// TIA Portal project "Mixing Fluid Projects" (V14)
// Project Files to accomodate the PLC Programming for Mixing Fluid Projects. 
// 
// PLEASE USE THE PROGRAM WISELY

(* hardware
DEVICE "S71500/ET200MP station_1"  S7-1500 station
   slot 0: "Rail_0"  Rack  6ES7 590-1***0-0AA0
   slot 0: "PS 60W 24/48/60VDC_1"  PS 60W 24/48/60VDC  6ES7 505-0RA00-0AB0  V1.0
   slot 1: "PLC_1"  CPU 1513-1 PN  6ES7 513-1AL01-0AB0  V2.1
      slot 3: "CPU display_1"  6ES7591-1AA00-0AA0
   slot 2: "DI 16x24VDC BA_1"  DI 16x24VDC BA  6ES7 521-1BH10-0AA0  V1.0
   slot 3: "DQ 16x24VDC/0.5A BA_1"  DQ 16x24VDC/0.5A BA  6ES7 522-1BH10-0AA0  V1.0
   slot 4: "AI 8xU/I/RTD/TC ST_1"  AI 8xU/I/RTD/TC ST  6ES7 531-7KF00-0AB0  V2.1
   slot 5: "AQ 8xU/I HS_1"  AQ 8xU/I HS  6ES7 532-5HF00-0AB0  V2.1
*)

// ===== PLC "PLC_1"  CPU 1513-1 PN =====

DATA_BLOCK "General_Tank Level_DB"   // DB4
{ S7_Optimized_Access := 'FALSE' }
VERSION : 0.1
   VAR
      "User Setpoint" : Int := 30;   // Setpoint Input from User
      PID_Level_Setpoint : Real;   // Setpoint into PID Level
      PID_Level_MV : Real;   // Output of PID Level (Manipulating Variable) on %
      PID_Level_MVNorm : Real;   // Output of PID Level (Manipulating Variable) on % Normalize
      PID_Level_MVInt : Int;   // Output of PID Level (Manipulating Variable) on % Integer
      PID_Level_ManualSlct : Bool;   // Switch for Activate Manual Mode
      PID_Level_InputMnlValue : Real;   // User Input Value for Manual MV
      PID_Level_ErrorAck : Bool;   // Acknowledged Button for Operator
      PID_Level_PIDReset : Bool;   // Reset Button for PID Compact
      PID_Level_ModeslctButton : Bool := true;   // Activate Mode Selection for PID Operation
      PID_Level_ModeValue : Int := 3;   // Select Mode for PID Operation from 1-4
      PID_Level_Alarm_SVHigh : Bool;   // Alarm from PID Level if Setpoint is Maximum
      PID_Level_Alarm_SVLow : Bool;   // Alarm from PID Level if Setpoint is Minimum
      PID_Level_Alarm_PVhigh : Bool;   // Alarm from PID Level if Process Value is Maximum
      PID_Level_Alarm_PVLow : Bool;   // Alarm from PID Level if Process Value is Minimum
      PID_Level_ModeStatus : Int;   // Status Mode for PID Operation
      PID_Level_ErrorStatus : Bool;   // Error Flag if PID Block is Occured
      PID_Level_ErrorBit : Real;   // Error Code if PID Block is Occured
      ControlValve_Level_Output : Real;   // Output of Level Control Valve
      ControlValve_Level_TravelMax : Bool;   // Level Control Valve Travel Max
      ControlValve_Level_TravelMin : Bool;   // Level Control Valve Travel Min
      "Level_Process Value" : Real := 50.0;   // Output from Level Process
      "Level_Process Reset" : Bool;   // Reset The Level Process
      Level_FlowarateAddRslt : Real;   // Additional PV from Hot + Cold Fluid Flowrate
      "Level_Flowrate Input" : Real;   // Total net flowrate going in/out from tank
      CascadeCommand : Bool;   // Command to activate Cascade PID Level Loop
      FeedforwardCmd : Bool;   // Command to activate Feedforward PID Level Loop
      LSH_Active : Bool;   // Alarm : Level Switch High Activate
      LSH_Warn : Bool;   // Alarm : Warning before LSH Active
      LSL_Active : Bool;   // Alarm : Level Switch Low Activate
      LSL_Warn : Bool;   // Alarm : Warning before LSL Active
      Trip_Reset : Bool := false;   // Alarm : Trip Command Reset
      PB_User : Real := 100.0;   // User Input for Proportional Band
      PB_UserDiv : Real := 0.0;   // User Input for Kp (Gain)
      Ti_User : Real := 104.7556;   // User Input for Integral Time
      Td_User : Real;   // User Input for Derivative Time
      SimpleFeedback_Status : Bool;   // Simple Feedback Loop Status Activate
   END_VAR
BEGIN
END_DATA_BLOCK

DATA_BLOCK "General_Flow Product 13_DB"   // DB5
{ S7_Optimized_Access := 'FALSE' }
VERSION : 0.1
   VAR
      User_Setpoint : Real := 2.0;   // Setpoint Input from User
      User_Setpoint_Norm : Real;   // Setpoint Input from User Normalized
      PID_Flow13_Setpoint : Real;   // Setpoint into PID Product Flowrate 13
      PID_Flow13_MV : Real;   // Output of PID Product Flowrate 13(Manipulating Variable) on %
      PID_Flow13_MVNorm : Real;   // Output of PID Product Flowrate 13(Manipulating Variable) on % Normalize
      PID_Flow13_MVInt : Int;   // Output of PID Product Flowrate 13 (Manipulating Variable) on % Integer
      PID_Flow13_ManualSlct : Bool;   // Switch for Activate Manual Mode
      PID_Flow13_InputMnlValue : Real;   // User Input Value for Manual MV
      PID_Flow13_ErrorAck : Bool;   // Acknowledged Button for Operator
      PID_Flow13_PIDReset : Bool;   // Reset Button for PID Compact
      PID_Flow13_ModeslctButton : Bool := true;   // Activate Mode Selection for PID Operation
      PID_Flow13_ModeValue : Int := 3;   // Select Mode for PID Operation from 1-4
      PID_Flow13_Alarm_SVHigh : Bool;   // Alarm from PID Product Flowrate 13 if Setpoint is Maximum
      PID_Flow13_Alarm_SVLow : Bool;   // Alarm from PID Product Flowrate 13 if Setpoint is Minimum
      PID_Flow13_Alarm_PVhigh : Bool;   // Alarm from PID Product Flowrate 13 if Process Value is Maximum
      PID_Flow13_Alarm_PVLow : Bool;   // Alarm from PID Product Flowrate 13 if Process Value is Minimum
      PID_Flow13_ModeStatus : Int;   // Status Mode for PID Operation
      PID_Flow13_ErrorStatus : Bool;   // Error Flag if PID Block is Occured
      PID_Flow13_ErrorBit : Real;   // Error Code if PID Block is Occured
      ControlValve_Flow13_Output : Real;   // Output of Product Flowrate 13 Control Valve
      ControlValve_Flow13_TravelMax : Bool;   // Product Flowrate 13 Control Valve Travel Max
      ControlValve_Flow13_TravelMin : Bool;   // Product Flowrate 13 Control Valve Travel Min
      "Flow13_Process Value" : Real;   // Output from Product Flowrate 13 Process
      "Flow13_Process ValueNorm" : Real;   // Output fromProduct Flowrate 13 Process Normalize
      "Flow13_Process Value_Status" : Real;   // Output Status from Product Flowrate
      "Flow13_Process Reset" : Bool;   // Reset The Product Flowrate 13Process
      SDV13_Active : Bool;   // Alarm : SDV13 Activate
      Pump13_CmdOffTrip : Bool;   // Turn off the Pump1-3 as Alarm Occured
      Pump13_CmdOff : Bool;   // Turn off the Pump1-3
      Pump13_CmdOn : Bool := false;   // Turn On the Pump1-3
      Pump13_Running : Bool := true;   // Pump1-3 Running Status
      Pump13_TripStatus : Bool;   // Pump1-3 Trip Status
      Pump13_TripReset : Bool := false;   // Pump1-3 Trip Reset Command
      PSL13_Active : Bool;   // Alarm : PSL Activate
      PSH13_Active : Bool;   // Alarm : PSH Activate
      PSH13_Reset : Bool;   // Reset Command of PSH13
      PB_User : Real := 21.71176;   // User Input for Proportional Band
      PB_UserDiv : Real;   // User Input for Kp (Gain)
      Ti_User : Real := 4.404553;   // User Input for Integral Time
      Td_User : Real := 0.0;   // User Input for Derivative Time
   END_VAR
BEGIN
END_DATA_BLOCK

DATA_BLOCK "General_Product Temperature_DB"   // DB9
{ S7_Optimized_Access := 'FALSE' }
VERSION : 0.1
   VAR
      User_Setpoint : Int := 40;   // Setpoint Input from User
      User_Setpoint_Norm : Real;   // Setpoint Input from User Normalized
      PID_Temp_Setpoint : Real;   // Setpoint into PID Product Temperature
      PID_Temp_MV : Real;   // Output of PID Product Temperature(Manipulating Variable) on %
      PID_Temp_MVNorm : Real;   // Output of PID Product Temperature(Manipulating Variable) on % Normalize
      PID_Temp_MVInt : Int;   // Output of PID Product Temperature (Manipulating Variable) on % Integer
      PID_Temp_ManualSlct : Bool;   // Switch for Activate Manual Mode
      PID_Temp_InputMnlValue : Real;   // User Input Value for Manual MV
      PID_Temp_ErrorAck : Bool;   // Acknowledged Button for Operator
      PID_Temp_PIDReset : Bool;   // Reset Button for PID Compact
      PID_Temp_ModeslctButton : Bool := true;   // Activate Mode Selection for PID Operation
      PID_Temp_ModeValue : Int := 3;   // Select Mode for PID Operation from 1-4
      PID_Temp_Alarm_SVHigh : Bool;   // Alarm from PID Product Temperature if Setpoint is Maximum
      PID_Temp_Alarm_SVLow : Bool;   // Alarm from PID Product Temperature if Setpoint is Minimum
      PID_Temp_Alarm_PVhigh : Bool;   // Alarm from PID Product Temperature if Process Value is Maximum
      PID_Temp_Alarm_PVLow : Bool;   // Alarm from PID Product Temperature if Process Value is Minimum
      PID_Temp_ModeStatus : Int;   // Status Mode for PID Operation
      PID_Temp_ErrorStatus : Bool;   // Error Flag if PID Block is Occured
      PID_Temp_ErrorBit : Real;   // Error Code if PID Block is Occured
      ControlValve_Temp_Output : Real;   // Output of Product Temperature Control Valve
      ControlValve_Temp_TravelMax : Bool;   // Product Temperature Control Valve Travel Max
      ControlValve_Temp_TravelMin : Bool;   // Product Temperature Control Valve Travel Min
      "Temp_Process Value" : Real;   // Output from Product Temperature Process
      "Temp_Process ValueRaw" : Real := 50.0;   // Output from Product Temperature Process raw
      "Temp_Process ValueNorm" : Real;   // Output fromProduct Temperature Process Normalize
      "Temp_Process Value_Status" : Real;   // Output Status from Product Temperature
      "Temp_Process Reset" : Bool;   // Reset The Product TemperatureProcess
      BlackCalc_HotFluid1Calc : Real;   // Hot Fluid Aspect Flowarate Heat released
      BlackCalc_ColdFluid1Calc_1 : Real;   // Hot Fluid Aspect Flowarate Heat received
      BlackCalc_Nominator : Real;   // Total additional of Black Calculation in Nominator
      BlackCalc_HotFluidFlowrate : Real;   // Flowrate of Hot Fluid in System
      BlackCalc_denominator : Real;   // Total additional of Black Calculation in denominator
      CascadeCmd : Bool;   // Cascade Command between Temp Product - Cold Fluid Flowrate
      FeedforwardCmd : Bool;   // Feedforward Command for Product Temp Control
      TSH_active : Bool;   // Alarm : Temp Switch High Activate
      TSH_Warn : Bool;   // Alarm : Warning before TSH Active
      TSL_active : Bool;   // Alarm : Temp Switch Low Activate
      TSL_Warn : Bool;   // Alarm : Warning before LSL Active
      Trip_Reset : Bool := false;   // Alarm : Trip Command Reset
      PB_User : Real := 50.0;   // User Input for Proportional Band
      PB_UserDiv : Real;   // User Input for Kp (Gain)
      Ti_User : Real := 4.404553;   // User Input for Integral Time
      Td_User : Real := 0.0;   // User Input for Derivative Time
      SimpleFeedback_Status : Bool;   // Simple Feedback Loop Status Activate
   END_VAR
BEGIN
END_DATA_BLOCK

DATA_BLOCK "General_Hot Fluid Flow_DB"   // DB12
{ S7_Optimized_Access := 'FALSE' }
VERSION : 0.1
   VAR
      User_Setpoint : Real := 2.5;   // Setpoint Input from User
      User_Setpoint_Norm : Real;   // Setpoint Input from User Normalized
      PID_Flow11_Setpoint : Real;   // Setpoint into PID Hot Fluid Flowrate
      PID_Flow11_MV : Real;   // Output of PIDHot Fluid Flowrate(Manipulating Variable) on %
      PID_Flow11_MVNorm : Real;   // Output of PID Hot Fluid Flowrate(Manipulating Variable) on % Normalize
      PID_Flow11_MVInt : Int;   // Output of PID Hot Fluid Flowrate (Manipulating Variable) on % Integer
      PID_Flow11_ManualSlct : Bool;   // Switch for Activate Manual Mode
      PID_Flow11_InputMnlValue : Real;   // User Input Value for Manual MV
      PID_Flow11_ErrorAck : Bool;   // Acknowledged Button for Operator
      PID_Flow11_PIDReset : Bool;   // Reset Button for PID Compact
      PID_Flow11_ModeslctButton : Bool := true;   // Activate Mode Selection for PID Operation
      PID_Flow11_ModeValue : Int := 3;   // Select Mode for PID Operation from 1-4
      PID_Flow11_Alarm_SVHigh : Bool;   // Alarm from PID Hot Fluid Flowrate if Setpoint is Maximum
      PID_Flow11_Alarm_SVLow : Bool;   // Alarm from PID Hot Fluid Flowrate if Setpoint is Minimum
      PID_Flow11_Alarm_PVhigh : Bool;   // Alarm from PID Hot Fluid Flowrate if Process Value is Maximum
      PID_Flow11_Alarm_PVLow : Bool;   // Alarm from PID Hot Fluid Flowrate if Process Value is Minimum
      PID_Flow11_ModeStatus : Int;   // Status Mode for PID Operation
      PID_Flow11_ErrorStatus : Bool;   // Error Flag if PID Block is Occured
      PID_Flow11_ErrorBit : Real;   // Error Code if PID Block is Occured
      ControlValve_Flow11_Output : Real;   // Output of Hot Fluid Flowrate Control Valve
      ControlValve_Flow11_TravelMax : Bool;   // Product Hot Fluid Flowrate Control Valve Travel Max
      ControlValve_Flow11_TravelMin : Bool;   // Product Hot Fluid Flowrate Control Valve Travel Min
      "Flow11_Process Value" : Real;   // Output from Hot Fluid Flowrate Process
      "Flow11_Process ValueNorm" : Real;   // Output fromHot Fluid Flowrate Process Normalize
      "Flow11_Process Value_Status" : Real;   // Output Status from Hot Fluid Flowrate
      "Flow11_Process Reset" : Bool;   // Reset The Hot Fluid Flowrate Process
      Flow11_LoopActv : Bool := true;   // Command to activate Hot Fluid Control Loop Only
      SDV11_Active : Bool;   // Alarm : SDV11_Activate
      Pump11_CmdOffTrip : Bool;   // Turn Off the Pump1-1 as Alarm Activate
      Pump11_CmdOff : Bool;   // Turn off the Pump1-1
      Pump11_CmdOn : Bool := false;   // Turn On the Pump1-1
      Pump11_Running : Bool := true;   // Pump1-1 Running Status
      Pump11_TripStatus : Bool;   // Pump1-1 Trip Status
      Pump11_TripReset : Bool := false;   // Pump1-1 Trip Reset Command
      PSL11_Active : Bool;   // Alarm : PSL Activate
      PSH11_Active : Bool;   // Alarm : PSH Activate
      PSH11_Reset : Bool := false;   // Reset Command of PSH11
      PB_User : Real := 100.0;   // User Input for Proportional Band
      PB_UserDiv : Real;   // User Input for Kp (Gain)
      Ti_User : Real := 20.0;   // User Input for Integral Time
      Td_User : Real;   // User Input for Derivative Time
   END_VAR
BEGIN
END_DATA_BLOCK

DATA_BLOCK "General_Cold Fluid Flow_DB"   // DB15
{ S7_Optimized_Access := 'FALSE' }
VERSION : 0.1
   VAR
      User_Setpoint : Real := 1.7;   // Setpoint Input from User
      User_Setpoint_Norm : Real;   // Setpoint Input from User Normalized
      PID_Flow12_Setpoint : Real;   // Setpoint into PID Cold Fluid Flowrate
      PID_Flow12_MV : Real;   // Output of PID Cold Fluid Flowrate(Manipulating Variable) on %
      PID_Flow12_MVNorm : Real;   // Output of PID Cold Fluid Flowrate(Manipulating Variable) on % Normalize
      PID_Flow12_MVInt : Int;   // Output of PID Cold Fluid Flowrate (Manipulating Variable) on % Integer
      PID_Flow12_ManualSlct : Bool;   // Switch for Activate Manual Mode
      PID_Flow12_InputMnlValue : Real;   // User Input Value for Manual MV
      PID_Flow12_ErrorAck : Bool;   // Acknowledged Button for Operator
      PID_Flow12_PIDReset : Bool;   // Reset Button for PID Compact
      PID_Flow12_ModeslctButton : Bool := true;   // Activate Mode Selection for PID Operation
      PID_Flow12_ModeValue : Int := 3;   // Select Mode for PID Operation from 1-4
      PID_Flow12_Alarm_SVHigh : Bool;   // Alarm from PID Cold Fluid Flowrate if Setpoint is Maximum
      PID_Flow12_Alarm_SVLow : Bool;   // Alarm from PID Cold Fluid Flowrate if Setpoint is Minimum
      PID_Flow12_Alarm_PVhigh : Bool;   // Alarm from PID ColdFluid Flowrate if Process Value is Maximum
      PID_Flow12_Alarm_PVLow : Bool;   // Alarm from PID Cold Fluid Flowrate if Process Value is Minimum
      PID_Flow12_ModeStatus : Int;   // Status Mode for PID Operation
      PID_Flow12_ErrorStatus : Bool;   // Error Flag if PID Block is Occured
      PID_Flow12_ErrorBit : Real;   // Error Code if PID Block is Occured
      ControlValve_Flow12_Output : Real;   // Output of Cold Fluid Flowrate Control Valve
      ControlValve_Flow12_TravelMax : Bool;   // Product Cold Fluid Flowrate Control Valve Travel Max
      ControlValve_Flow12_TravelMin : Bool;   // Product Cold Fluid Flowrate Control Valve Travel Min
      "Flow12_Process Value" : Real;   // Output from Cold Fluid Flowrate Process
      "Flow12_Process ValueNorm" : Real;   // Output from Cold Fluid Flowrate Process Normalize
      "Flow12_Process Value_Status" : Real;   // Output Status from Cold Fluid Flowrate
      "Flow12_Process Reset" : Bool;   // Reset The Cold Fluid Flowrate Process
      Flow12_LoopActv : Bool := true;   // Activate the Cold Fluid Control Loop Only
      SDV12_Active : Bool;   // Alarm : SDV12 activate
      Pump12_CmdOffTrip : Bool;   // Turn Off the Pump1-2 as Alarm Occured
      Pump12_CmdOff : Bool;   // Turn off the Pump1-2
      Pump12_CmdOn : Bool := false;   // Turn On the Pump1-2
      Pump12_Running : Bool := true;   // Pump1-2 Running Status
      Pump12_TripStatus : Bool;   // Pump1-2 Trip Status
      Pump12_TripReset : Bool := false;   // Pump1-2 Trip Reset Command
      PSL12_Active : Bool;   // Alarm : PSL Activate
      PSH12_Active : Bool;   // Alarm : PSH Activate
      PSH12_Reset : Bool;   // Reset Command of PSH12
      PB_User : Real := 21.56999;   // User Input for Proportional Band
      PB_UserDiv : Real;   // User Input for Kp (Gain)
      Ti_User : Real := 4.443021;   // User Input for Integral Time
      Td_User : Real := 0.0;   // User Input for Derivative Time
   END_VAR
BEGIN
END_DATA_BLOCK

// folder: Alarm Group DB

DATA_BLOCK "Program Alarm_DB_LSH"   // DB22
{ S7_Optimized_Access := 'TRUE' }
VERSION : 0.1
// stored: InstanceOfName Program Alarm
"Program Alarm"
BEGIN
END_DATA_BLOCK

DATA_BLOCK "Program Alarm_DB_LSL"   // DB23
{ S7_Optimized_Access := 'TRUE' }
VERSION : 0.1
// stored: InstanceOfName Program Alarm
"Program Alarm"
BEGIN
END_DATA_BLOCK

DATA_BLOCK "Program Alarm Unack_DB_LSHWarn"   // DB24
{ S7_Optimized_Access := 'TRUE' }
VERSION : 0.1
// stored: InstanceOfName Program Alarm Unack
"Program Alarm Unack"
BEGIN
END_DATA_BLOCK

DATA_BLOCK "Program Alarm Unack_DB_LSLWarn"   // DB25
{ S7_Optimized_Access := 'TRUE' }
VERSION : 0.1
// stored: InstanceOfName Program Alarm Unack
"Program Alarm Unack"
BEGIN
END_DATA_BLOCK

DATA_BLOCK "Program Alarm_DB_TSH"   // DB26
{ S7_Optimized_Access := 'TRUE' }
VERSION : 0.1
// stored: InstanceOfName Program Alarm
"Program Alarm"
BEGIN
END_DATA_BLOCK

DATA_BLOCK "Program Alarm Unack_DB_TSHWarn"   // DB27
{ S7_Optimized_Access := 'TRUE' }
VERSION : 0.1
// stored: InstanceOfName Program Alarm Unack
"Program Alarm Unack"
BEGIN
END_DATA_BLOCK

DATA_BLOCK "Program Alarm_DB_TSL"   // DB28
{ S7_Optimized_Access := 'TRUE' }
VERSION : 0.1
// stored: InstanceOfName Program Alarm
"Program Alarm"
BEGIN
END_DATA_BLOCK

DATA_BLOCK "Program Alarm Unack_DB_TSLWarn"   // DB29
{ S7_Optimized_Access := 'TRUE' }
VERSION : 0.1
// stored: InstanceOfName Program Alarm Unack
"Program Alarm Unack"
BEGIN
END_DATA_BLOCK

DATA_BLOCK "Program Alarm_DB_PSH11"   // DB30
{ S7_Optimized_Access := 'TRUE' }
VERSION : 0.1
// stored: InstanceOfName Program Alarm
"Program Alarm"
BEGIN
END_DATA_BLOCK

DATA_BLOCK "Program Alarm_DB_SDV11"   // DB31
{ S7_Optimized_Access := 'TRUE' }
VERSION : 0.1
// stored: InstanceOfName Program Alarm
"Program Alarm"
BEGIN
END_DATA_BLOCK

DATA_BLOCK "Program Alarm_DB_Pump11TripStatus"   // DB32
{ S7_Optimized_Access := 'TRUE' }
VERSION : 0.1
// stored: InstanceOfName Program Alarm
"Program Alarm"
BEGIN
END_DATA_BLOCK

DATA_BLOCK "Program Alarm Unack_DB_Pump11Run"   // DB33
{ S7_Optimized_Access := 'TRUE' }
VERSION : 0.1
// stored: InstanceOfName Program Alarm Unack
"Program Alarm Unack"
BEGIN
END_DATA_BLOCK

DATA_BLOCK "Program Alarm Unack_DB_Pump11CmdOff"   // DB34
{ S7_Optimized_Access := 'TRUE' }
VERSION : 0.1
// stored: InstanceOfName Program Alarm Unack
"Program Alarm Unack"
BEGIN
END_DATA_BLOCK

DATA_BLOCK "Program Alarm Unack_DB_Pump11TripReset"   // DB35
{ S7_Optimized_Access := 'TRUE' }
VERSION : 0.1
// stored: InstanceOfName Program Alarm Unack
"Program Alarm Unack"
BEGIN
END_DATA_BLOCK

DATA_BLOCK "Program Alarm Unack_DB_PSL11"   // DB36
{ S7_Optimized_Access := 'TRUE' }
VERSION : 0.1
// stored: InstanceOfName Program Alarm Unack
"Program Alarm Unack"
BEGIN
END_DATA_BLOCK

DATA_BLOCK "Program Alarm Unack_DB_PSH11Reset"   // DB37
{ S7_Optimized_Access := 'TRUE' }
VERSION : 0.1
// stored: InstanceOfName Program Alarm Unack
"Program Alarm Unack"
BEGIN
END_DATA_BLOCK

DATA_BLOCK "Program Alarm_DB_PSH12"   // DB38
{ S7_Optimized_Access := 'TRUE' }
VERSION : 0.1
// stored: InstanceOfName Program Alarm
"Program Alarm"
BEGIN
END_DATA_BLOCK

DATA_BLOCK "Program Alarm_DB_SDV12"   // DB39
{ S7_Optimized_Access := 'TRUE' }
VERSION : 0.1
// stored: InstanceOfName Program Alarm
"Program Alarm"
BEGIN
END_DATA_BLOCK

DATA_BLOCK "Program Alarm_DB_Pump12TripStatus"   // DB40
{ S7_Optimized_Access := 'TRUE' }
VERSION : 0.1
// stored: InstanceOfName Program Alarm
"Program Alarm"
BEGIN
END_DATA_BLOCK

DATA_BLOCK "Program Alarm Unack_DB_Pump12Run"   // DB41
{ S7_Optimized_Access := 'TRUE' }
VERSION : 0.1
// stored: InstanceOfName Program Alarm Unack
"Program Alarm Unack"
BEGIN
END_DATA_BLOCK

DATA_BLOCK "Program Alarm Unack_DB_Pump12CmdOff"   // DB42
{ S7_Optimized_Access := 'TRUE' }
VERSION : 0.1
// stored: InstanceOfName Program Alarm Unack
"Program Alarm Unack"
BEGIN
END_DATA_BLOCK

DATA_BLOCK "Program Alarm Unack_DB_Pump12TripReset"   // DB43
{ S7_Optimized_Access := 'TRUE' }
VERSION : 0.1
// stored: InstanceOfName Program Alarm Unack
"Program Alarm Unack"
BEGIN
END_DATA_BLOCK

DATA_BLOCK "Program Alarm Unack_DB_PSL12"   // DB44
{ S7_Optimized_Access := 'TRUE' }
VERSION : 0.1
// stored: InstanceOfName Program Alarm Unack
"Program Alarm Unack"
BEGIN
END_DATA_BLOCK

DATA_BLOCK "Program Alarm Unack_DB_PSH12Reset"   // DB45
{ S7_Optimized_Access := 'TRUE' }
VERSION : 0.1
// stored: InstanceOfName Program Alarm Unack
"Program Alarm Unack"
BEGIN
END_DATA_BLOCK

DATA_BLOCK "Program Alarm_DB_PSH13"   // DB46
{ S7_Optimized_Access := 'TRUE' }
VERSION : 0.1
// stored: InstanceOfName Program Alarm
"Program Alarm"
BEGIN
END_DATA_BLOCK

DATA_BLOCK "Program Alarm_DB_SDV13"   // DB47
{ S7_Optimized_Access := 'TRUE' }
VERSION : 0.1
// stored: InstanceOfName Program Alarm
"Program Alarm"
BEGIN
END_DATA_BLOCK

DATA_BLOCK "Program Alarm_DB_Pump13TripStatus"   // DB48
{ S7_Optimized_Access := 'TRUE' }
VERSION : 0.1
// stored: InstanceOfName Program Alarm
"Program Alarm"
BEGIN
END_DATA_BLOCK

DATA_BLOCK "Program Alarm Unack_DB_Pump13Run"   // DB49
{ S7_Optimized_Access := 'TRUE' }
VERSION : 0.1
// stored: InstanceOfName Program Alarm Unack
"Program Alarm Unack"
BEGIN
END_DATA_BLOCK

DATA_BLOCK "Program Alarm Unack_DB_Pump13CmdOff"   // DB50
{ S7_Optimized_Access := 'TRUE' }
VERSION : 0.1
// stored: InstanceOfName Program Alarm Unack
"Program Alarm Unack"
BEGIN
END_DATA_BLOCK

DATA_BLOCK "Program Alarm Unack_DB_Pump13TripReset"   // DB51
{ S7_Optimized_Access := 'TRUE' }
VERSION : 0.1
// stored: InstanceOfName Program Alarm Unack
"Program Alarm Unack"
BEGIN
END_DATA_BLOCK

DATA_BLOCK "Program Alarm Unack_DB-PSL13"   // DB52
{ S7_Optimized_Access := 'TRUE' }
VERSION : 0.1
// stored: InstanceOfName Program Alarm Unack
"Program Alarm Unack"
BEGIN
END_DATA_BLOCK

DATA_BLOCK "Program Alarm Unack_DB_PSH13Reset"   // DB53
{ S7_Optimized_Access := 'TRUE' }
VERSION : 0.1
// stored: InstanceOfName Program Alarm Unack
"Program Alarm Unack"
BEGIN
END_DATA_BLOCK

DATA_BLOCK "Program Alarm Unack_DB_Level_Alarm Reset"   // DB54
{ S7_Optimized_Access := 'TRUE' }
VERSION : 0.1
// stored: InstanceOfName Program Alarm Unack
"Program Alarm Unack"
BEGIN
END_DATA_BLOCK

DATA_BLOCK "Program Alarm Unack_DB_Temp_Trip Reset"   // DB55
{ S7_Optimized_Access := 'TRUE' }
VERSION : 0.1
// stored: InstanceOfName Program Alarm Unack
"Program Alarm Unack"
BEGIN
END_DATA_BLOCK

// folder: System blocks/Program resources

DATA_BLOCK "Time On Delay PSH11"   // DB18
{ S7_Optimized_Access := 'TRUE' }
AUTHOR : Simatic
FAMILY : IEC
NAME : IEC_TMR
VERSION : 1.0
// stored: InstanceOfName IEC_TIMER
"IEC_TIMER"
BEGIN
END_DATA_BLOCK

DATA_BLOCK "Time On Delay PSH12"   // DB19
{ S7_Optimized_Access := 'TRUE' }
AUTHOR : Simatic
FAMILY : IEC
NAME : IEC_TMR
VERSION : 1.0
// stored: InstanceOfName IEC_TIMER
"IEC_TIMER"
BEGIN
END_DATA_BLOCK

DATA_BLOCK "Time On Delay PSH13"   // DB20
{ S7_Optimized_Access := 'TRUE' }
AUTHOR : Simatic
FAMILY : IEC
NAME : IEC_TMR
VERSION : 1.0
// stored: InstanceOfName IEC_TIMER
"IEC_TIMER"
BEGIN
END_DATA_BLOCK

DATA_BLOCK "TON_LSH"   // DB21
{ S7_Optimized_Access := 'TRUE' }
AUTHOR : Simatic
FAMILY : IEC
NAME : IEC_LTMR
VERSION : 1.0
// stored: InstanceOfName IEC_LTIMER
"IEC_LTIMER"
BEGIN
END_DATA_BLOCK

DATA_BLOCK "TON_LSL"   // DB56
{ S7_Optimized_Access := 'TRUE' }
AUTHOR : Simatic
FAMILY : IEC
NAME : IEC_LTMR
VERSION : 1.0
// stored: InstanceOfName IEC_LTIMER
"IEC_LTIMER"
BEGIN
END_DATA_BLOCK

DATA_BLOCK "TON_TSH"   // DB57
{ S7_Optimized_Access := 'TRUE' }
AUTHOR : Simatic
FAMILY : IEC
NAME : IEC_LTMR
VERSION : 1.0
// stored: InstanceOfName IEC_LTIMER
"IEC_LTIMER"
BEGIN
END_DATA_BLOCK

DATA_BLOCK "TON_TSL"   // DB58
{ S7_Optimized_Access := 'TRUE' }
AUTHOR : Simatic
FAMILY : IEC
NAME : IEC_TMR
VERSION : 1.0
// stored: InstanceOfName IEC_TIMER
"IEC_TIMER"
BEGIN
END_DATA_BLOCK

// folder: Utilities Group DB

DATA_BLOCK "Level Control Valve_DB"   // DB2
{ S7_Optimized_Access := 'TRUE' }
VERSION : 2.01
// stored: InstanceOfName LSim_Level Control Valve
"LSim_Level Control Valve"
BEGIN
   perOn := true;
END_DATA_BLOCK

DATA_BLOCK "LSim_Tank Process_DB"   // DB3
{ S7_Optimized_Access := 'TRUE' }
VERSION : 2.01
// stored: InstanceOfName LSim_Level Process
"LSim_Level Process"
BEGIN
END_DATA_BLOCK

DATA_BLOCK "Flow Control Valve 13_DB"   // DB7
{ S7_Optimized_Access := 'TRUE' }
VERSION : 2.01
// stored: InstanceOfName LSim_Flow Control Valve 13
"LSim_Flow Control Valve 13"
BEGIN
   perOn := true;
END_DATA_BLOCK

DATA_BLOCK "LSim_Product Flow 13 Process_DB"   // DB8
{ S7_Optimized_Access := 'TRUE' }
VERSION : 2.01
// stored: InstanceOfName LSim_Product Flowrate 13
"LSim_Product Flowrate 13"
BEGIN
END_DATA_BLOCK

DATA_BLOCK "LSim_Product Temp_DB"   // DB11
{ S7_Optimized_Access := 'TRUE' }
VERSION : 2.01
// stored: InstanceOfName LSim_Product Temp
"LSim_Product Temp"
BEGIN
   perOn := true;
END_DATA_BLOCK

DATA_BLOCK "LSim_Hot Fluid Flow_DB"   // DB14
{ S7_Optimized_Access := 'TRUE' }
VERSION : 2.01
// stored: InstanceOfName LSim_Hot Fluid Flowrate
"LSim_Hot Fluid Flowrate"
BEGIN
END_DATA_BLOCK

DATA_BLOCK "LSim_Cold Fluid Flowrate"   // DB17
{ S7_Optimized_Access := 'TRUE' }
VERSION : 2.01
// stored: InstanceOfName LSim_Cold Fluid Flow
"LSim_Cold Fluid Flow"
BEGIN
END_DATA_BLOCK

// folder: (top level)

FUNCTION_BLOCK "LSim_Flow Control Valve 13"   // FB1, FBD
{ S7_Optimized_Access := 'TRUE' }
VERSION : 2.01
// //============================================================================
// //SIEMENS AG
// //(c)Copyright 2017 All Rights Reserved
// //-----------------------------------------------------------------------------
// //Library:       Library for Controlled System Simulation
// //Tested with:   S7-1500 FW V2.0 / S7-1200 FW V4.2
// //Engineering:   STEP 7 V14 Upd2 (TIA Portal)
// //Restrictions:  Cyclic interrupt
// //Requirements:  memory card needed for S7-1500
// //Functionality: Simulation of a valve with adjustable transition time
// //-----------------------------------------------------------------------------
// //Change log table:
// //Version    Date             Expert in charge                               Changes applied
// //02.00.00 03.02.2016 Siemens Industry Online Support Release (STEP 7 V13 SP1)
// //02.00.01 02.03.2017 Siemens Industry Online Support Release (STEP 7 V14)
// //============================================================================
   VAR_INPUT
      inputUp : Bool := false;   // control signal “Open valve”
      inputDn : Bool := false;   // control signal “Close valve”
      inputPer : Int;   // Analog manipulated variable
      perOn : Bool;   // selection switch, whether inputUp/inputDn or inputPer is used (inputPer is used for TRUE)
      perMax : Real := 27648.0;   // upper limit of the analog value of the valve position.
      perMin : Real;   // lower limit of the analog value of the valve position
      realMax : Real := 100.0;   // upper limit of the converted floating-point value for the valve position
      realMin : Real;   // lower limit of the converted floating-point value for the valve position
      transitTime : Real := 20.0;   // traversing time of the value between the end positions
      cycle : Real := 0.1;   // cyclic time [sec]
      reset : Bool := false;   // resets all relevant parameters to ‘0’ including the output
   END_VAR
   VAR_OUTPUT
      output : Real := 0.0;   // calculated valve position (within the “realMin” and “realMax” limits)
      outputPer : Int;   // calculated analog valve position (within the “perMin” and “perMax” limits)
      highLimit : Bool := false;   // simulated upper valve end position reached at highLimit = TRUE
      lowLimit : Bool := false;   // simulated lower valve end position reached at lowLimit = TRUE
   END_VAR
   VAR
      statInput : Real;
      statDelta : Real;
      statOut : Real;
      statHigh : Bool;
      statLow : Bool;
   END_VAR
   VAR_TEMP
      tempReal : Real;
      tempStepWidth : Real;
      tempStepWidthNeg : Real;
      tempBool : Bool;
      tempInputNorm : Real;
      tempUpFlag : Bool;
      tempDnFlag : Bool;
      tempInt : Int;
   END_VAR
   VAR_TEMP   // added for the SCL form of the ladder/FBD networks
      _w1 : Bool;
   END_VAR
BEGIN

REGION Network 1: reset
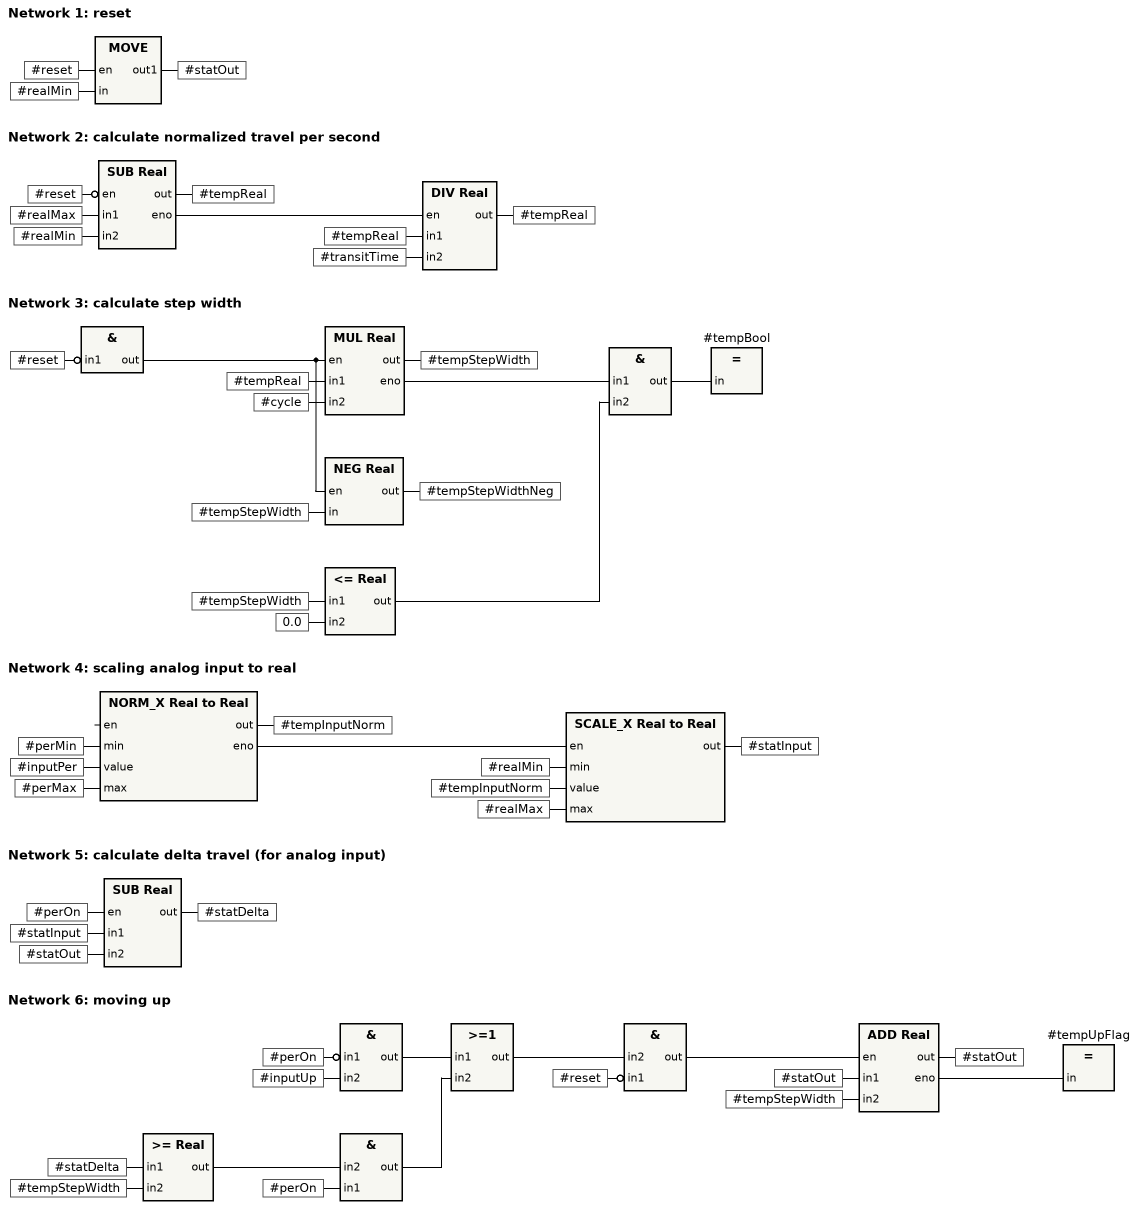
   IF #reset THEN #statOut := #realMin; END_IF;
END_REGION

REGION Network 2: calculate normalized travel per second
   // ENO of a box is taken as its EN; it also drops when the box reports an error
   IF NOT #reset THEN
       #tempReal := #realMax - #realMin;
       #tempReal := #tempReal / #transitTime;
   END_IF;
END_REGION

REGION Network 3: calculate step width
   // ENO of a box is taken as its EN; it also drops when the box reports an error
   IF NOT #reset THEN #tempStepWidth := #tempReal * #cycle; END_IF;
   #tempBool := NOT #reset AND (#tempStepWidth <= 0.0);
   IF NOT #reset THEN #tempStepWidthNeg := -#tempStepWidth; END_IF;
END_REGION

REGION Network 4: scaling analog input to real
   // ENO of a box is taken as its EN; it also drops when the box reports an error
   #tempInputNorm := NORM_X(MIN := #perMin, VALUE := #inputPer, MAX := #perMax);
   #statInput := SCALE_X(MIN := #realMin, VALUE := #tempInputNorm, MAX := #realMax);
END_REGION

REGION Network 5: calculate delta travel (for analog input)
   IF #perOn THEN #statDelta := #statInput - #statOut; END_IF;
END_REGION

REGION Network 6: moving up
   // ENO of a box is taken as its EN; it also drops when the box reports an error
   #_w1 := ((NOT #perOn AND #inputUp) OR ((#statDelta >= #tempStepWidth) AND #perOn)) AND NOT #reset;
   IF #_w1 THEN #statOut := #statOut + #tempStepWidth; END_IF;
   #tempUpFlag := #_w1;
END_REGION

REGION Network 7: checking max. limit
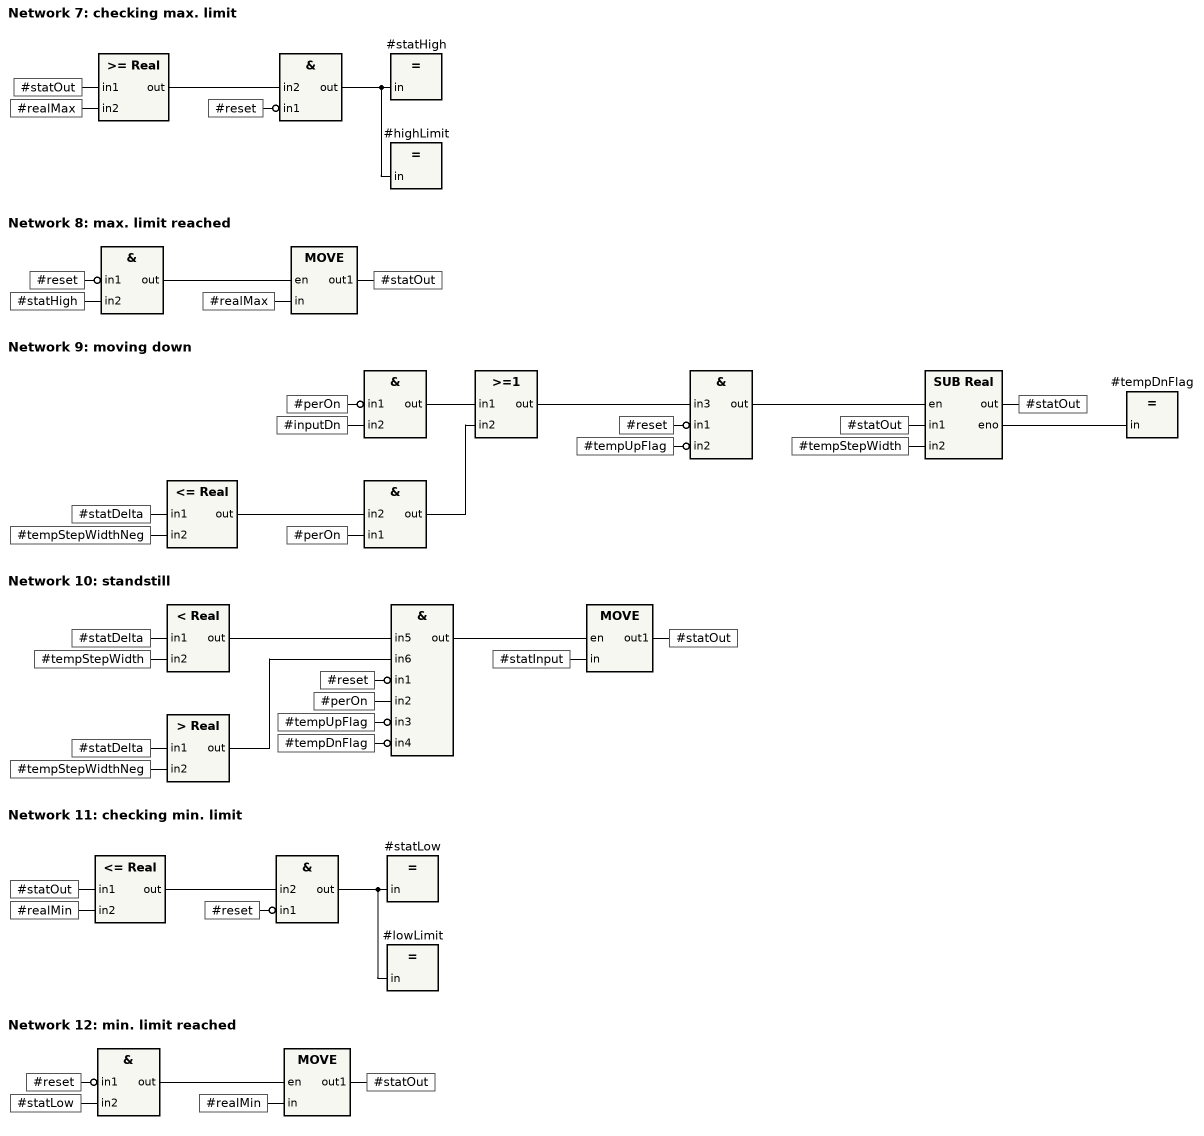
   #statHigh := (#statOut >= #realMax) AND NOT #reset;
   #highLimit := #statHigh;
END_REGION

REGION Network 8: max. limit reached
   IF NOT #reset AND #statHigh THEN #statOut := #realMax; END_IF;
END_REGION

REGION Network 9: moving down
   // ENO of a box is taken as its EN; it also drops when the box reports an error
   #_w1 := ((NOT #perOn AND #inputDn) OR ((#statDelta <= #tempStepWidthNeg) AND #perOn)) AND NOT #reset AND NOT #tempUpFlag;
   IF #_w1 THEN #statOut := #statOut - #tempStepWidth; END_IF;
   #tempDnFlag := #_w1;
END_REGION

REGION Network 10: standstill
   IF (#statDelta < #tempStepWidth) AND (#statDelta > #tempStepWidthNeg) AND NOT #reset AND #perOn AND NOT #tempUpFlag AND NOT #tempDnFlag THEN
       #statOut := #statInput;
   END_IF;
END_REGION

REGION Network 11: checking min. limit
   #statLow := (#statOut <= #realMin) AND NOT #reset;
   #lowLimit := #statLow;
END_REGION

REGION Network 12: min. limit reached
   IF NOT #reset AND #statLow THEN #statOut := #realMin; END_IF;
END_REGION

REGION Network 13: output and scaling to analog
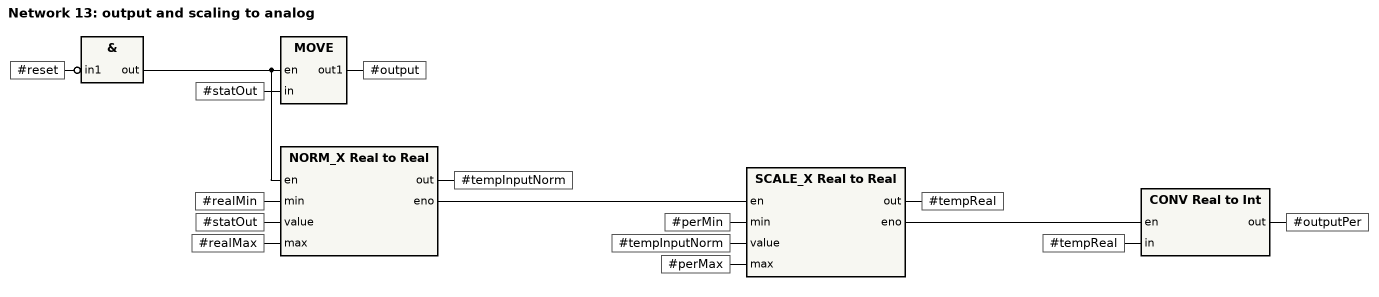
   // ENO of a box is taken as its EN; it also drops when the box reports an error
   IF NOT #reset THEN
       #output := #statOut;
       #tempInputNorm := NORM_X(MIN := #realMin, VALUE := #statOut, MAX := #realMax);
       #tempReal := SCALE_X(MIN := #perMin, VALUE := #tempInputNorm, MAX := #perMax);
       #outputPer := REAL_TO_INT(#tempReal);
   END_IF;
END_REGION
END_FUNCTION_BLOCK

FUNCTION_BLOCK "LSim_Product Temp"   // FB2, FBD
{ S7_Optimized_Access := 'TRUE' }
VERSION : 2.01
// //============================================================================
// //SIEMENS AG
// //(c)Copyright 2017 All Rights Reserved
// //-----------------------------------------------------------------------------
// //Library:       Library for Controlled System Simulation
// //Tested with:   S7-1500 FW V2.0 / S7-1200 FW V4.2
// //Engineering:   STEP 7 V14 Upd2 (TIA Portal)
// //Restrictions:  Cyclic interrupt
// //Requirements:  memory card needed for S7-1500
// //Functionality: Simulation of a valve with adjustable transition time
// //-----------------------------------------------------------------------------
// //Change log table:
// //Version    Date             Expert in charge                               Changes applied
// //02.00.00 03.02.2016 Siemens Industry Online Support Release (STEP 7 V13 SP1)
// //02.00.01 02.03.2017 Siemens Industry Online Support Release (STEP 7 V14)
// //============================================================================
   VAR_INPUT
      inputUp : Bool := false;   // control signal “Open valve”
      inputDn : Bool := false;   // control signal “Close valve”
      inputPer : Int;   // Analog manipulated variable
      perOn : Bool;   // selection switch, whether inputUp/inputDn or inputPer is used (inputPer is used for TRUE)
      perMax : Real := 27648.0;   // upper limit of the analog value of the valve position.
      perMin : Real;   // lower limit of the analog value of the valve position
      realMax : Real := 100.0;   // upper limit of the converted floating-point value for the valve position
      realMin : Real;   // lower limit of the converted floating-point value for the valve position
      transitTime : Real := 20.0;   // traversing time of the value between the end positions
      cycle : Real := 0.1;   // cyclic time [sec]
      reset : Bool := false;   // resets all relevant parameters to ‘0’ including the output
   END_VAR
   VAR_OUTPUT
      output : Real := 0.0;   // calculated valve position (within the “realMin” and “realMax” limits)
      outputPer : Int;   // calculated analog valve position (within the “perMin” and “perMax” limits)
      highLimit : Bool := false;   // simulated upper valve end position reached at highLimit = TRUE
      lowLimit : Bool := false;   // simulated lower valve end position reached at lowLimit = TRUE
   END_VAR
   VAR
      statInput : Real;
      statDelta : Real;
      statOut : Real;
      statHigh : Bool;
      statLow : Bool;
   END_VAR
   VAR_TEMP
      tempReal : Real;
      tempStepWidth : Real;
      tempStepWidthNeg : Real;
      tempBool : Bool;
      tempInputNorm : Real;
      tempUpFlag : Bool;
      tempDnFlag : Bool;
      tempInt : Int;
   END_VAR
   VAR_TEMP   // added for the SCL form of the ladder/FBD networks
      _w1 : Bool;
   END_VAR
BEGIN

REGION Network 1: reset
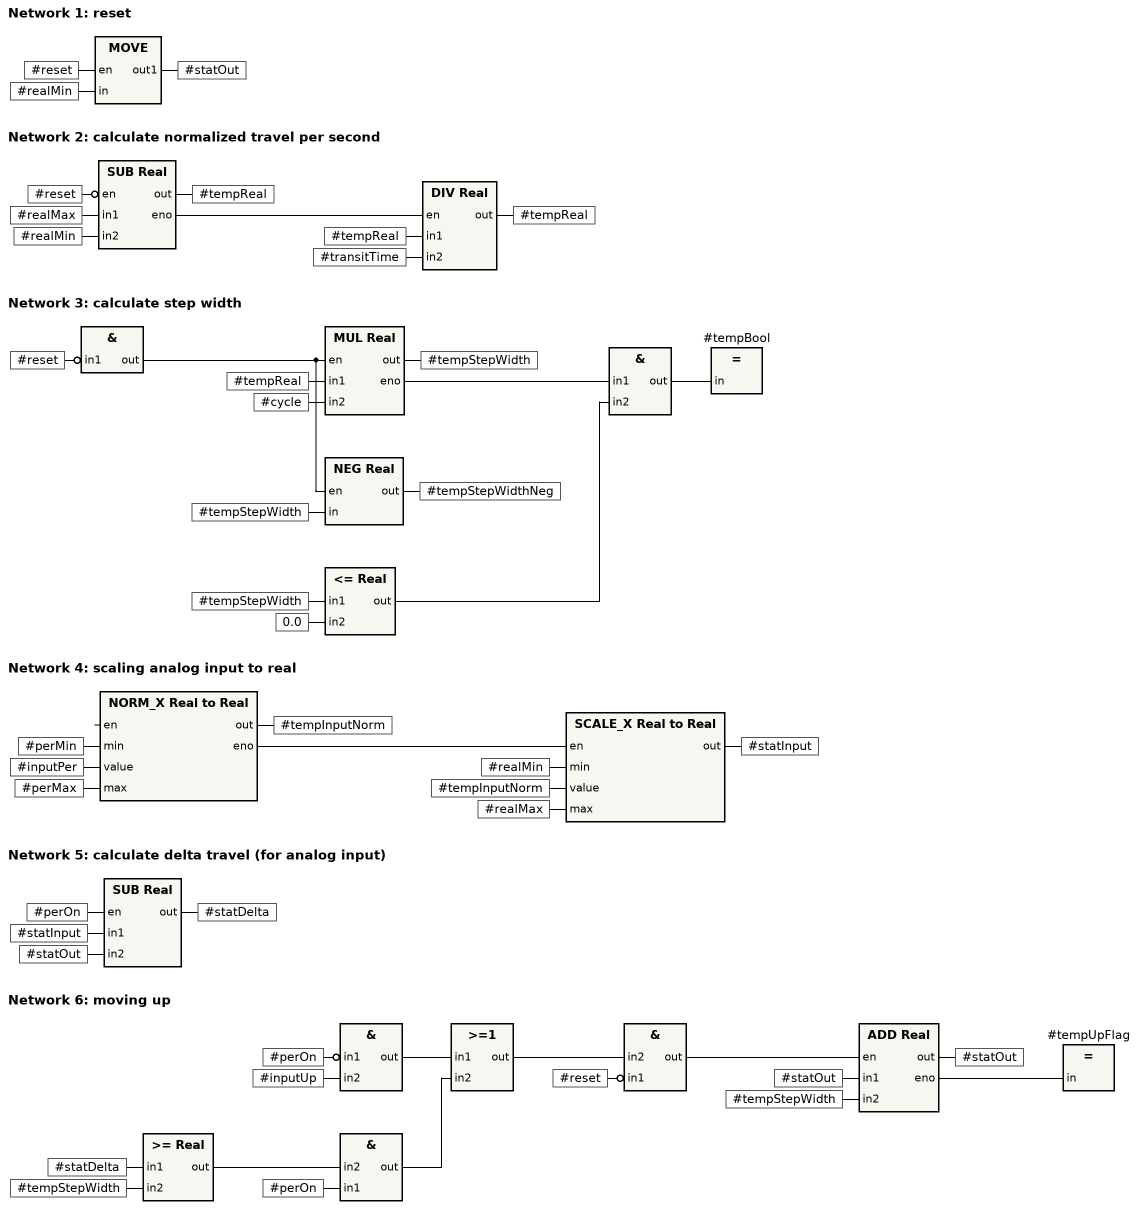
   IF #reset THEN #statOut := #realMin; END_IF;
END_REGION

REGION Network 2: calculate normalized travel per second
   // ENO of a box is taken as its EN; it also drops when the box reports an error
   IF NOT #reset THEN
       #tempReal := #realMax - #realMin;
       #tempReal := #tempReal / #transitTime;
   END_IF;
END_REGION

REGION Network 3: calculate step width
   // ENO of a box is taken as its EN; it also drops when the box reports an error
   IF NOT #reset THEN #tempStepWidth := #tempReal * #cycle; END_IF;
   #tempBool := NOT #reset AND (#tempStepWidth <= 0.0);
   IF NOT #reset THEN #tempStepWidthNeg := -#tempStepWidth; END_IF;
END_REGION

REGION Network 4: scaling analog input to real
   // ENO of a box is taken as its EN; it also drops when the box reports an error
   #tempInputNorm := NORM_X(MIN := #perMin, VALUE := #inputPer, MAX := #perMax);
   #statInput := SCALE_X(MIN := #realMin, VALUE := #tempInputNorm, MAX := #realMax);
END_REGION

REGION Network 5: calculate delta travel (for analog input)
   IF #perOn THEN #statDelta := #statInput - #statOut; END_IF;
END_REGION

REGION Network 6: moving up
   // ENO of a box is taken as its EN; it also drops when the box reports an error
   #_w1 := ((NOT #perOn AND #inputUp) OR ((#statDelta >= #tempStepWidth) AND #perOn)) AND NOT #reset;
   IF #_w1 THEN #statOut := #statOut + #tempStepWidth; END_IF;
   #tempUpFlag := #_w1;
END_REGION

REGION Network 7: checking max. limit
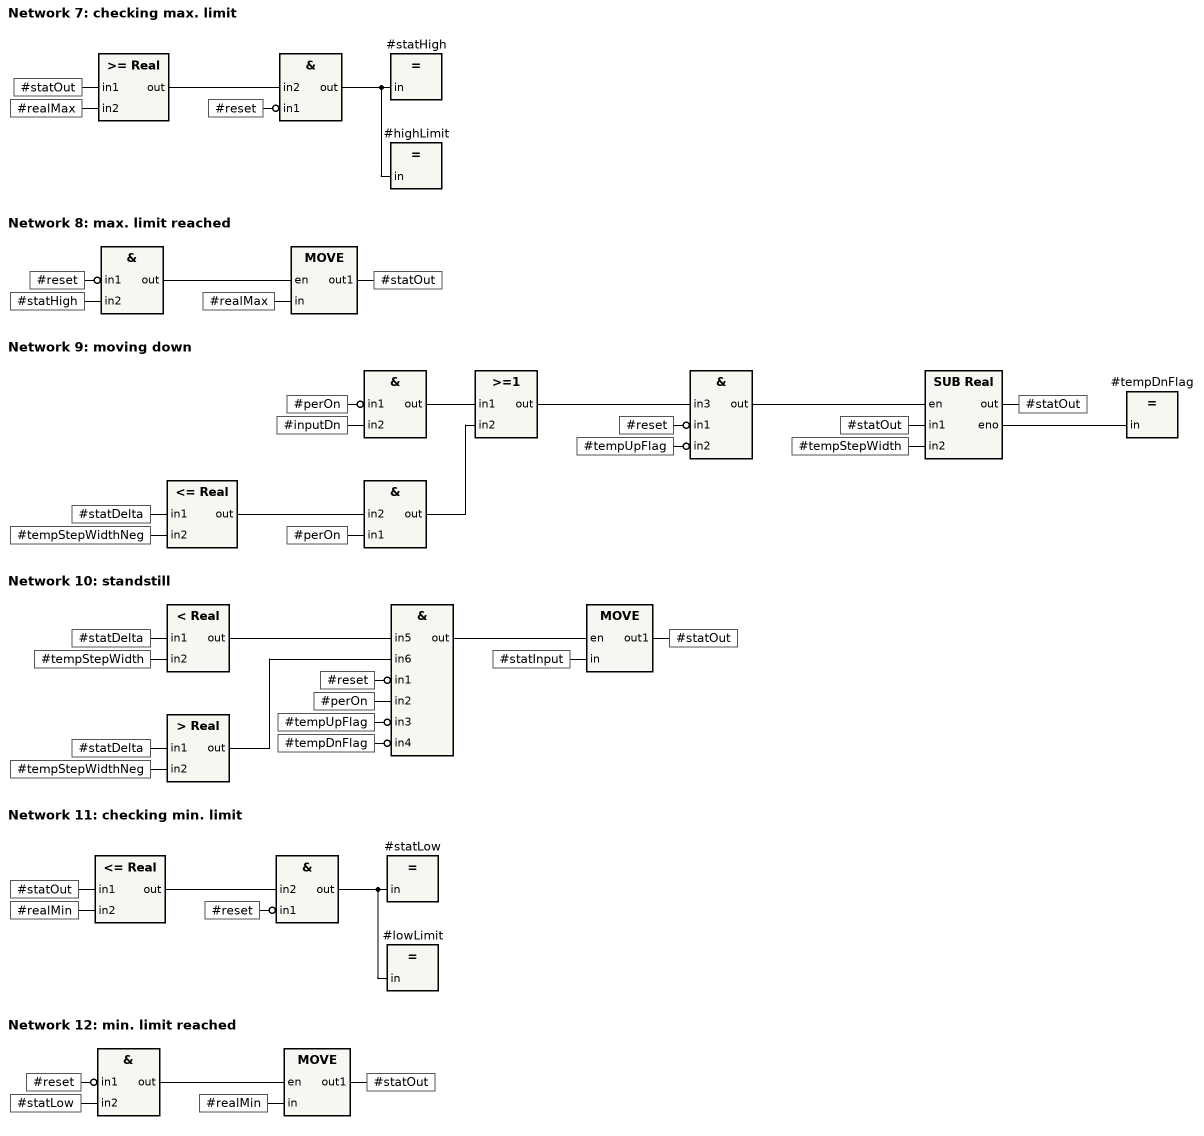
   #statHigh := (#statOut >= #realMax) AND NOT #reset;
   #highLimit := #statHigh;
END_REGION

REGION Network 8: max. limit reached
   IF NOT #reset AND #statHigh THEN #statOut := #realMax; END_IF;
END_REGION

REGION Network 9: moving down
   // ENO of a box is taken as its EN; it also drops when the box reports an error
   #_w1 := ((NOT #perOn AND #inputDn) OR ((#statDelta <= #tempStepWidthNeg) AND #perOn)) AND NOT #reset AND NOT #tempUpFlag;
   IF #_w1 THEN #statOut := #statOut - #tempStepWidth; END_IF;
   #tempDnFlag := #_w1;
END_REGION

REGION Network 10: standstill
   IF (#statDelta < #tempStepWidth) AND (#statDelta > #tempStepWidthNeg) AND NOT #reset AND #perOn AND NOT #tempUpFlag AND NOT #tempDnFlag THEN
       #statOut := #statInput;
   END_IF;
END_REGION

REGION Network 11: checking min. limit
   #statLow := (#statOut <= #realMin) AND NOT #reset;
   #lowLimit := #statLow;
END_REGION

REGION Network 12: min. limit reached
   IF NOT #reset AND #statLow THEN #statOut := #realMin; END_IF;
END_REGION

REGION Network 13: output and scaling to analog
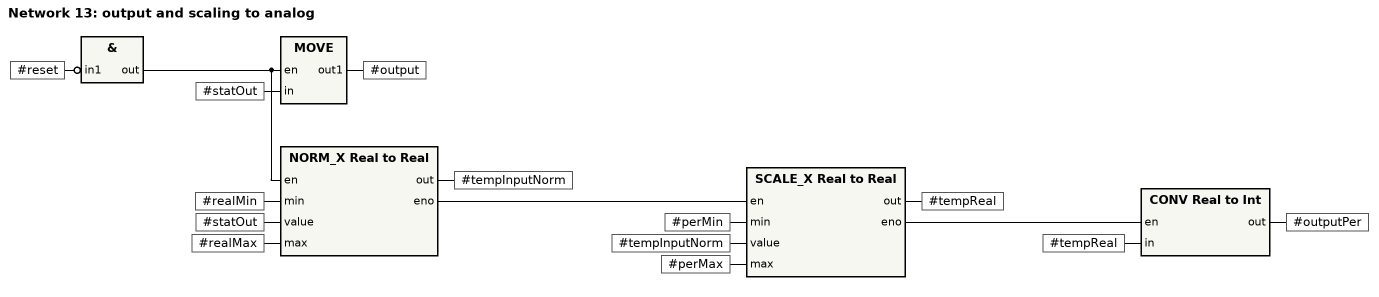
   // ENO of a box is taken as its EN; it also drops when the box reports an error
   IF NOT #reset THEN
       #output := #statOut;
       #tempInputNorm := NORM_X(MIN := #realMin, VALUE := #statOut, MAX := #realMax);
       #tempReal := SCALE_X(MIN := #perMin, VALUE := #tempInputNorm, MAX := #perMax);
       #outputPer := REAL_TO_INT(#tempReal);
   END_IF;
END_REGION
END_FUNCTION_BLOCK

FUNCTION_BLOCK "LSim_Hot Fluid Flowrate"   // FB3, SCL
{ S7_Optimized_Access := 'TRUE' }
VERSION : 2.01
   VAR_INPUT
      calcParam : Bool;   // recalculate with new parameters
      input : Real;   // input signal
      tmLag1 : Real := 1.0;   // time constant T1 [sec]
      gain : Real := 1.0;   // gain factor
      cycle : Real := 0.1;   // cyclic time [sec]
      maxOut : Real := 100.0;   // max. output limit
      minOut : Real;   // min. output limit
      reset : Bool;   // resets all relevant parameters to ‘0’ including the output
   END_VAR
   VAR_OUTPUT
      error : Bool;   // error (#tmLag1 <= 0)
      status : Word;   // status (if #tmLag1 <= 0 then status = 16#8001)
      maxReached : Bool;   // output has reached max. limit
      minReached : Bool;   // output has reached min. limit
      output : Real;   // output signal (if #error = FALSE)
   END_VAR
   VAR
      statRf1 : Real;
      statRe1 : Real;
      statOverfirst : Bool;
      statOutput : Real;
   END_VAR
BEGIN
   //=============================================================================
   //SIEMENS AG
   //(c)Copyright 2017 All Rights Reserved
   //-----------------------------------------------------------------------------
   //Library:       Library for Controlled System Simulation
   //Tested with:   S7-1500 FW V2.0 / S7-1200 FW V4.2
   //Engineering:   STEP 7 V14 Upd2 (TIA Portal)
   //Restrictions:  Cyclic interrupt
   //Requirements:  memory card needed for S7-1500
   //Functionality: Simulation of a PT1-System
   //
   //              gain
   //  F(p) = ---------------
   //          tmLag1 * p + 1
   //          
   //  Call the simulation in a cyclic interrupt with
   //  cyclic interrupt time at least = tmLag1/10!
   //-----------------------------------------------------------------------------
   //Change log table:
   //Version  Date       Expert in charge                Changes applied
   //02.00.00 03.02.2016 Siemens Industry Online Support Release (STEP 7 V13 SP1)
   //02.00.01 02.03.2017 Siemens Industry Online Support Release (STEP 7 V14)
   //=============================================================================
   // check parameter
   IF #tmLag1 <= 0 THEN
     #error := TRUE;
     #status := W#16#8001;     // Parameter Error
     #statOutput := 0;
     #output := 0;
     RETURN;
   ELSE
     #error := FALSE;
     #status := W#16#0000;     // no error
   END_IF;

   IF #calcParam = True OR NOT #statOverfirst THEN
     #statOverfirst:=1;
   // Z-parameters For Laplace PT1-System
   #statRe1 := - EXP(-#cycle/#tmLag1);
   #statRf1 := #gain*(1 + #statRe1);
   END_IF;

   // Differencial Equation of PT1-System
   #statOutput := #input*#statRf1 - #statOutput*#statRe1;

   // max limit of acutating variable
   IF #statOutput > #maxOut THEN
     #statOutput := #maxOut;
     #maxReached:= True;
   ELSE
     #maxReached := False;
   END_IF;

   // min limit of acutating variable
   IF #statOutput < #minOut THEN
     #statOutput := #minOut;
     #minReached := True;
   ELSE
     #minReached := False;
   END_IF;

   IF #reset THEN
     #statOutput := 0;
   END_IF;

   #output := #statOutput;
END_FUNCTION_BLOCK

FUNCTION_BLOCK "LSim_Cold Fluid Flow"   // FB4, SCL
{ S7_Optimized_Access := 'TRUE' }
VERSION : 2.01
   VAR_INPUT
      calcParam : Bool;   // recalculate with new parameters
      input : Real;   // input signal
      tmLag1 : Real := 1.0;   // time constant T1 [sec]
      gain : Real := 1.0;   // gain factor
      cycle : Real := 0.1;   // cyclic time [sec]
      maxOut : Real := 100.0;   // max. output limit
      minOut : Real;   // min. output limit
      reset : Bool;   // resets all relevant parameters to ‘0’ including the output
   END_VAR
   VAR_OUTPUT
      error : Bool;   // error (#tmLag1 <= 0)
      status : Word;   // status (if #tmLag1 <= 0 then status = 16#8001)
      maxReached : Bool;   // output has reached max. limit
      minReached : Bool;   // output has reached min. limit
      output : Real;   // output signal (if #error = FALSE)
   END_VAR
   VAR
      statRf1 : Real;
      statRe1 : Real;
      statOverfirst : Bool;
      statOutput : Real;
   END_VAR
BEGIN
   //=============================================================================
   //SIEMENS AG
   //(c)Copyright 2017 All Rights Reserved
   //-----------------------------------------------------------------------------
   //Library:       Library for Controlled System Simulation
   //Tested with:   S7-1500 FW V2.0 / S7-1200 FW V4.2
   //Engineering:   STEP 7 V14 Upd2 (TIA Portal)
   //Restrictions:  Cyclic interrupt
   //Requirements:  memory card needed for S7-1500
   //Functionality: Simulation of a PT1-System
   //
   //              gain
   //  F(p) = ---------------
   //          tmLag1 * p + 1
   //          
   //  Call the simulation in a cyclic interrupt with
   //  cyclic interrupt time at least = tmLag1/10!
   //-----------------------------------------------------------------------------
   //Change log table:
   //Version  Date       Expert in charge                Changes applied
   //02.00.00 03.02.2016 Siemens Industry Online Support Release (STEP 7 V13 SP1)
   //02.00.01 02.03.2017 Siemens Industry Online Support Release (STEP 7 V14)
   //=============================================================================
   // check parameter
   IF #tmLag1 <= 0 THEN
     #error := TRUE;
     #status := W#16#8001;     // Parameter Error
     #statOutput := 0;
     #output := 0;
     RETURN;
   ELSE
     #error := FALSE;
     #status := W#16#0000;     // no error
   END_IF;

   IF #calcParam = True OR NOT #statOverfirst THEN
     #statOverfirst:=1;
   // Z-parameters For Laplace PT1-System
   #statRe1 := - EXP(-#cycle/#tmLag1);
   #statRf1 := #gain*(1 + #statRe1);
   END_IF;

   // Differencial Equation of PT1-System
   #statOutput := #input*#statRf1 - #statOutput*#statRe1;

   // max limit of acutating variable
   IF #statOutput > #maxOut THEN
     #statOutput := #maxOut;
     #maxReached:= True;
   ELSE
     #maxReached := False;
   END_IF;

   // min limit of acutating variable
   IF #statOutput < #minOut THEN
     #statOutput := #minOut;
     #minReached := True;
   ELSE
     #minReached := False;
   END_IF;

   IF #reset THEN
     #statOutput := 0;
   END_IF;

   #output := #statOutput;
END_FUNCTION_BLOCK

FUNCTION_BLOCK "Program Alarm"   // FB6, LAD
{ S7_Optimized_Access := 'TRUE' }
VERSION : 0.1
   VAR_INPUT
      AlarmInput : Bool;
      Tag : String;
      AlarmText : String;
   END_VAR
   VAR
      "Program_Alarm_Level System" : Program_Alarm;
   END_VAR
   VAR_TEMP
      Error : Bool;
      Status : Word;
   END_VAR
BEGIN

REGION Network 1
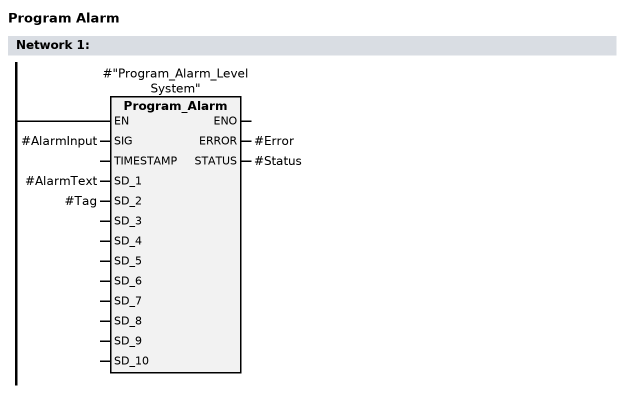
   #"Program_Alarm_Level System"(SIG := #AlarmInput,   // Program_Alarm
                           SD_1 := #AlarmText,
                           SD_2 := #Tag,
                           Error => #Error,
                           Status => #Status);
END_REGION
END_FUNCTION_BLOCK

FUNCTION_BLOCK "Program Alarm Unack"   // FB7, LAD
TITLE = UnAcknowledge Alarm Program
{ S7_Optimized_Access := 'TRUE' }
VERSION : 0.1
// Program for UnAcknowledged Alarm Data Block
   VAR_INPUT
      Alarminput : Bool;
      tag : String;
      alarmtext : String;
   END_VAR
   VAR
      Program_Alarm_Unack : Program_Alarm;
   END_VAR
   VAR_TEMP
      Error : Bool;
      Status : Word;
   END_VAR
BEGIN

REGION Network 1: UnAcknowledge Alarm Program
   // Program for UnAcknowledged Alarm Data Block
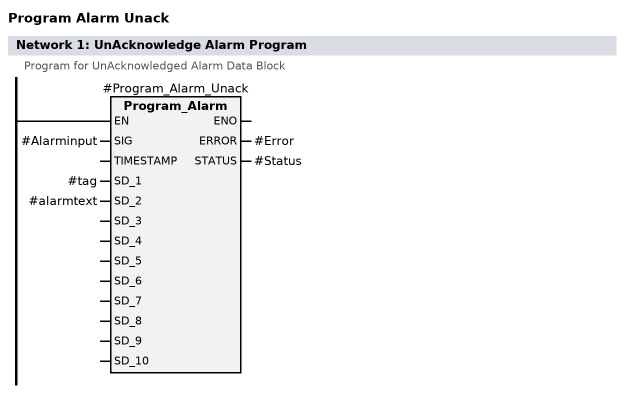
   #Program_Alarm_Unack(SIG := #Alarminput,   // Program_Alarm
                        SD_1 := #tag,
                        SD_2 := #alarmtext,
                        Error => #Error,
                        Status => #Status);
END_REGION
END_FUNCTION_BLOCK

FUNCTION_BLOCK "LSim_Product Flowrate 13"   // FB50, SCL
{ S7_Optimized_Access := 'TRUE' }
VERSION : 2.01
   VAR_INPUT
      calcParam : Bool;   // recalculate with new parameters
      input : Real;   // input signal
      tmLag1 : Real := 1.0;   // time constant T1 [sec]
      gain : Real := 1.0;   // gain factor
      cycle : Real := 0.1;   // cyclic time [sec]
      maxOut : Real := 100.0;   // max. output limit
      minOut : Real;   // min. output limit
      reset : Bool;   // resets all relevant parameters to ‘0’ including the output
   END_VAR
   VAR_OUTPUT
      error : Bool;   // error (#tmLag1 <= 0)
      status : Word;   // status (if #tmLag1 <= 0 then status = 16#8001)
      maxReached : Bool;   // output has reached max. limit
      minReached : Bool;   // output has reached min. limit
      output : Real;   // output signal (if #error = FALSE)
   END_VAR
   VAR
      statRf1 : Real;
      statRe1 : Real;
      statOverfirst : Bool;
      statOutput : Real;
   END_VAR
BEGIN
   //=============================================================================
   //SIEMENS AG
   //(c)Copyright 2017 All Rights Reserved
   //-----------------------------------------------------------------------------
   //Library:       Library for Controlled System Simulation
   //Tested with:   S7-1500 FW V2.0 / S7-1200 FW V4.2
   //Engineering:   STEP 7 V14 Upd2 (TIA Portal)
   //Restrictions:  Cyclic interrupt
   //Requirements:  memory card needed for S7-1500
   //Functionality: Simulation of a PT1-System
   //
   //              gain
   //  F(p) = ---------------
   //          tmLag1 * p + 1
   //          
   //  Call the simulation in a cyclic interrupt with
   //  cyclic interrupt time at least = tmLag1/10!
   //-----------------------------------------------------------------------------
   //Change log table:
   //Version  Date       Expert in charge                Changes applied
   //02.00.00 03.02.2016 Siemens Industry Online Support Release (STEP 7 V13 SP1)
   //02.00.01 02.03.2017 Siemens Industry Online Support Release (STEP 7 V14)
   //=============================================================================
   // check parameter
   IF #tmLag1 <= 0 THEN
     #error := TRUE;
     #status := W#16#8001;     // Parameter Error
     #statOutput := 0;
     #output := 0;
     RETURN;
   ELSE
     #error := FALSE;
     #status := W#16#0000;     // no error
   END_IF;

   IF #calcParam = True OR NOT #statOverfirst THEN
     #statOverfirst:=1;
   // Z-parameters For Laplace PT1-System
   #statRe1 := - EXP(-#cycle/#tmLag1);
   #statRf1 := #gain*(1 + #statRe1);
   END_IF;

   // Differencial Equation of PT1-System
   #statOutput := #input*#statRf1 - #statOutput*#statRe1;

   // max limit of acutating variable
   IF #statOutput > #maxOut THEN
     #statOutput := #maxOut;
     #maxReached:= True;
   ELSE
     #maxReached := False;
   END_IF;

   // min limit of acutating variable
   IF #statOutput < #minOut THEN
     #statOutput := #minOut;
     #minReached := True;
   ELSE
     #minReached := False;
   END_IF;

   IF #reset THEN
     #statOutput := 0;
   END_IF;

   #output := #statOutput;
END_FUNCTION_BLOCK

FUNCTION_BLOCK "LSim_Level Process"   // FB56, SCL
{ S7_Optimized_Access := 'TRUE' }
VERSION : 2.01
   VAR_INPUT
      calcParam : Bool;   // recalculate with new parameters
      input : Real;   // input signal
      tmLag1 : Real := 1.0;   // time constant T1 [sec]
      cycle : Real := 0.1;   // cyclic time [sec]
      maxOut : Real := 100.0;   // max. output limit
      minOut : Real;   // min. output limit
      reset : Bool;   // resets all relevant parameters to ‘0’ including the output
   END_VAR
   VAR_OUTPUT
      error : Bool;   // error (#tmLag1 <= 0)
      status : Word;   // status (if #tmLag1 <= 0 then status = 16#8001)
      maxReached : Bool;   // output has reached max. limit
      minReached : Bool;   // output has reached min. limit
      output : Real;   // output signal (if #error = FALSE)
   END_VAR
   VAR
      statRxn1 : Real;   // delayed input signal (n-1)
      statRyn1 : Real;   // delayed output signal (n-1)
      statRa1 : Real;
      statRb1 : Real;
      statOverfirst : Bool;
      statOutput : Real;   // output signal
   END_VAR
BEGIN
   //=============================================================================
   //SIEMENS AG
   //(c)Copyright 2017 All Rights Reserved
   //-----------------------------------------------------------------------------
   //Library:       Library for Controlled System Simulation
   //Tested with:   S7-1500 FW V2.0 / S7-1200 FW V4.2
   //Engineering:   STEP 7 V14 Upd2 (TIA Portal)
   //Restrictions:  Cyclic interrupt
   //Requirements:  memory card needed for S7-1500
   //Functionality: Simulation of a I-System
   //
   //             1
   //  F(p) = -----------
   //         (tmLag1*p)
   //          
   //  Call the simulation in a cyclic interrupt with
   //  cyclic interrupt time at least = tmLag1/10!
   //-----------------------------------------------------------------------------
   //Change log table:
   //Version  Date       Expert in charge                Changes applied
   //02.00.00 03.02.2016 Siemens Industry Online Support Release (STEP 7 V13 SP1)
   //02.00.01 02.03.2017 Siemens Industry Online Support Release (STEP 7 V14)
   //=============================================================================

   // check parameter
   IF #tmLag1 <= 0 THEN
     #error := True;
     #status := W#16#8001;     // Parameter Error
     #statRxn1 := 0.0;
     #statRyn1 := 0.0;
     #statOutput := 0;
     #output := 0;
     RETURN;
   ELSE
     #error := FALSE;
     #status := W#16#0000;     // no error
   END_IF;

   // calculates the z-parameter for the difference equatation
   IF #calcParam = True OR NOT #statOverfirst THEN
   #statOverfirst:=1;
     // Calculate z-parameters for IT1-System
   #statRb1 := #cycle/#tmLag1;
   #statRa1 := -1;

   END_IF;

   // reset Memory
   IF #reset = True THEN
     #statRxn1 := 0.0;
     #statRyn1 := 0.0;
     #statOutput:=0;
   END_IF;

   // save delayed output-signals
   #statRyn1:= #statOutput;

   // difference equatation for the I-system
   #statOutput := #statRxn1* #statRb1 - #statRyn1*#statRa1;

   // save delayed input-signals
   #statRxn1 := #input;

   // max limit of acutating variable
   IF #statOutput > #maxOut THEN
     #statOutput := #maxOut;
     #maxReached:= True;
   ELSE
     #maxReached := False;
   END_IF;

   // min limit of acutating variable
   IF #statOutput < #minOut THEN
     #statOutput := #minOut;
     #minReached := True;
   ELSE
     #minReached := False;
   END_IF;

   #output := #statOutput;
END_FUNCTION_BLOCK

FUNCTION_BLOCK "LSim_Level Control Valve"   // FB63, FBD
{ S7_Optimized_Access := 'TRUE' }
VERSION : 2.01
// //============================================================================
// //SIEMENS AG
// //(c)Copyright 2017 All Rights Reserved
// //-----------------------------------------------------------------------------
// //Library:       Library for Controlled System Simulation
// //Tested with:   S7-1500 FW V2.0 / S7-1200 FW V4.2
// //Engineering:   STEP 7 V14 Upd2 (TIA Portal)
// //Restrictions:  Cyclic interrupt
// //Requirements:  memory card needed for S7-1500
// //Functionality: Simulation of a valve with adjustable transition time
// //-----------------------------------------------------------------------------
// //Change log table:
// //Version    Date             Expert in charge                               Changes applied
// //02.00.00 03.02.2016 Siemens Industry Online Support Release (STEP 7 V13 SP1)
// //02.00.01 02.03.2017 Siemens Industry Online Support Release (STEP 7 V14)
// //============================================================================
   VAR_INPUT
      inputUp : Bool := false;   // control signal “Open valve”
      inputDn : Bool := false;   // control signal “Close valve”
      inputPer : Int;   // Analog manipulated variable
      perOn : Bool;   // selection switch, whether inputUp/inputDn or inputPer is used (inputPer is used for TRUE)
      perMax : Real := 27648.0;   // upper limit of the analog value of the valve position.
      perMin : Real;   // lower limit of the analog value of the valve position
      realMax : Real := 100.0;   // upper limit of the converted floating-point value for the valve position
      realMin : Real;   // lower limit of the converted floating-point value for the valve position
      transitTime : Real := 20.0;   // traversing time of the value between the end positions
      cycle : Real := 0.1;   // cyclic time [sec]
      reset : Bool := false;   // resets all relevant parameters to ‘0’ including the output
   END_VAR
   VAR_OUTPUT
      output : Real := 0.0;   // calculated valve position (within the “realMin” and “realMax” limits)
      outputPer : Int;   // calculated analog valve position (within the “perMin” and “perMax” limits)
      highLimit : Bool := false;   // simulated upper valve end position reached at highLimit = TRUE
      lowLimit : Bool := false;   // simulated lower valve end position reached at lowLimit = TRUE
   END_VAR
   VAR
      statInput : Real;
      statDelta : Real;
      statOut : Real;
      statHigh : Bool;
      statLow : Bool;
   END_VAR
   VAR_TEMP
      tempReal : Real;
      tempStepWidth : Real;
      tempStepWidthNeg : Real;
      tempBool : Bool;
      tempInputNorm : Real;
      tempUpFlag : Bool;
      tempDnFlag : Bool;
      tempInt : Int;
   END_VAR
   VAR_TEMP   // added for the SCL form of the ladder/FBD networks
      _w1 : Bool;
   END_VAR
BEGIN

REGION Network 1: reset
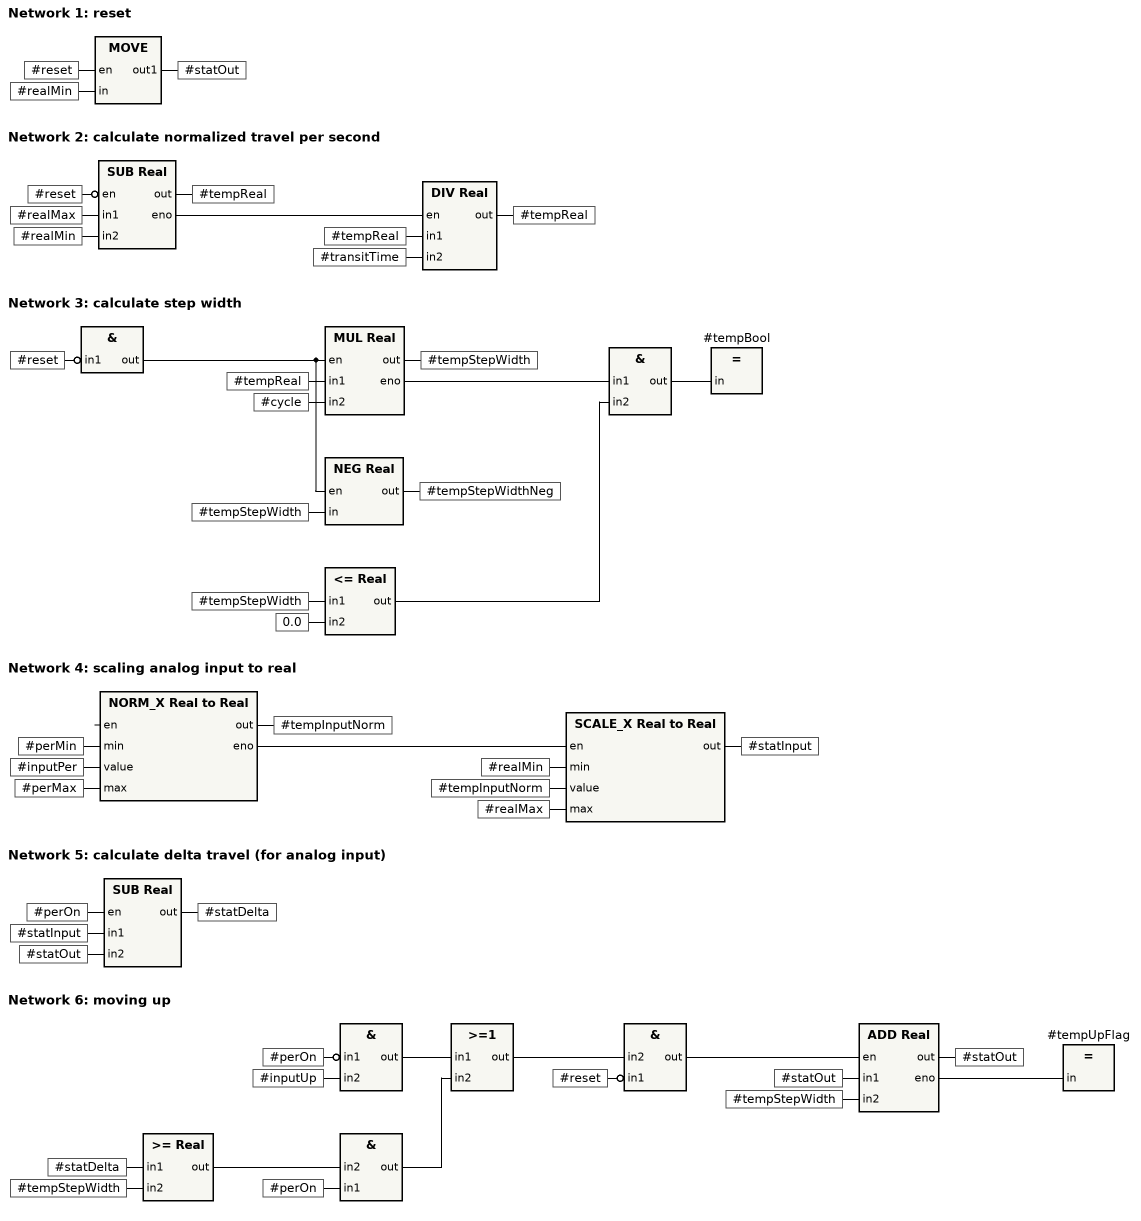
   IF #reset THEN #statOut := #realMin; END_IF;
END_REGION

REGION Network 2: calculate normalized travel per second
   // ENO of a box is taken as its EN; it also drops when the box reports an error
   IF NOT #reset THEN
       #tempReal := #realMax - #realMin;
       #tempReal := #tempReal / #transitTime;
   END_IF;
END_REGION

REGION Network 3: calculate step width
   // ENO of a box is taken as its EN; it also drops when the box reports an error
   IF NOT #reset THEN #tempStepWidth := #tempReal * #cycle; END_IF;
   #tempBool := NOT #reset AND (#tempStepWidth <= 0.0);
   IF NOT #reset THEN #tempStepWidthNeg := -#tempStepWidth; END_IF;
END_REGION

REGION Network 4: scaling analog input to real
   // ENO of a box is taken as its EN; it also drops when the box reports an error
   #tempInputNorm := NORM_X(MIN := #perMin, VALUE := #inputPer, MAX := #perMax);
   #statInput := SCALE_X(MIN := #realMin, VALUE := #tempInputNorm, MAX := #realMax);
END_REGION

REGION Network 5: calculate delta travel (for analog input)
   IF #perOn THEN #statDelta := #statInput - #statOut; END_IF;
END_REGION

REGION Network 6: moving up
   // ENO of a box is taken as its EN; it also drops when the box reports an error
   #_w1 := ((NOT #perOn AND #inputUp) OR ((#statDelta >= #tempStepWidth) AND #perOn)) AND NOT #reset;
   IF #_w1 THEN #statOut := #statOut + #tempStepWidth; END_IF;
   #tempUpFlag := #_w1;
END_REGION

REGION Network 7: checking max. limit
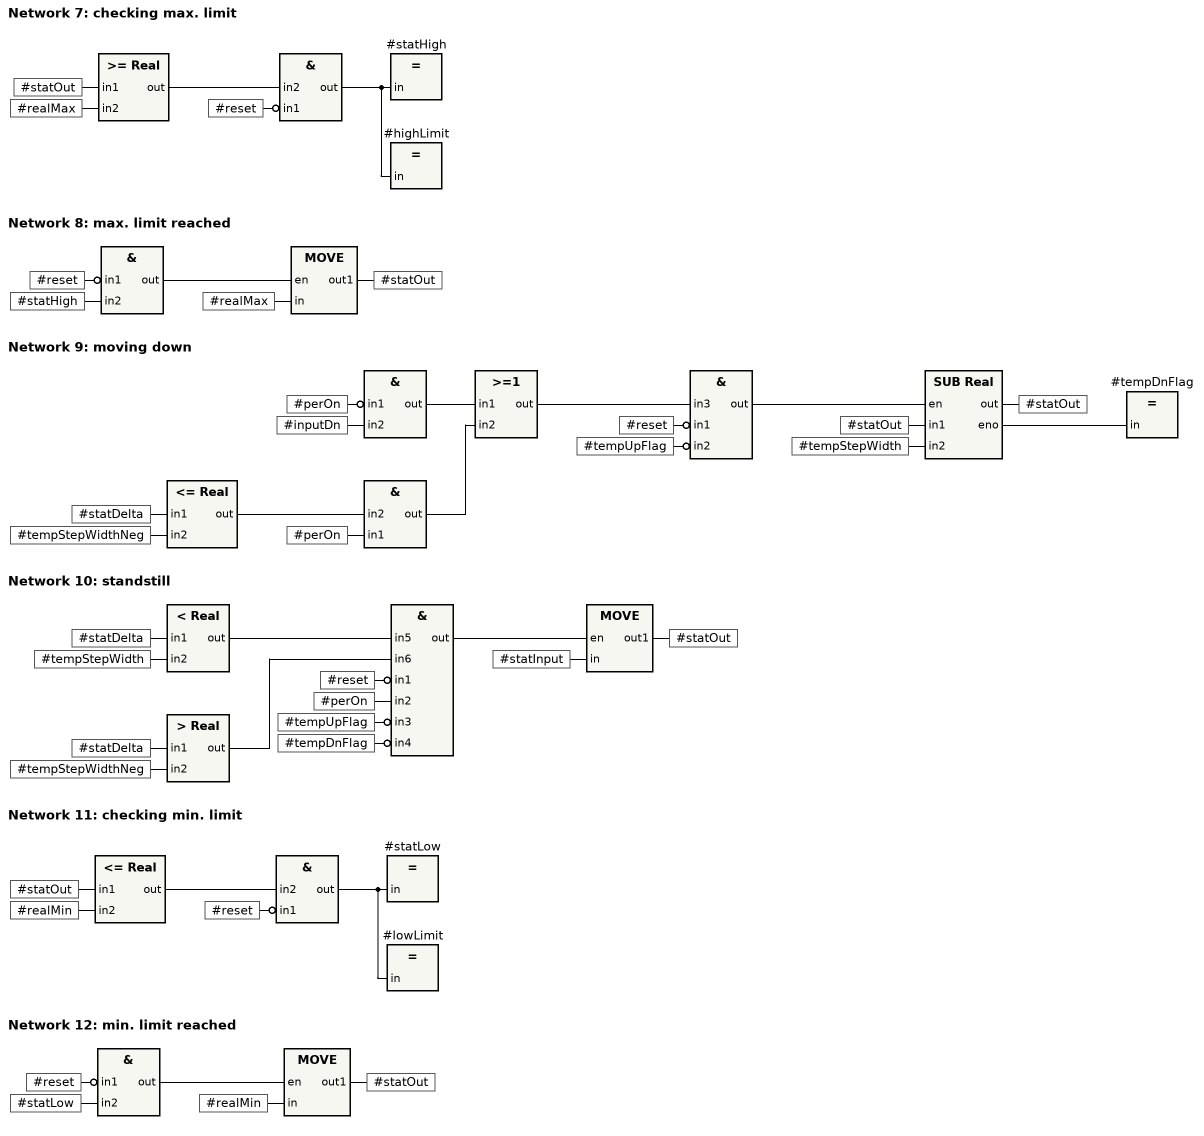
   #statHigh := (#statOut >= #realMax) AND NOT #reset;
   #highLimit := #statHigh;
END_REGION

REGION Network 8: max. limit reached
   IF NOT #reset AND #statHigh THEN #statOut := #realMax; END_IF;
END_REGION

REGION Network 9: moving down
   // ENO of a box is taken as its EN; it also drops when the box reports an error
   #_w1 := ((NOT #perOn AND #inputDn) OR ((#statDelta <= #tempStepWidthNeg) AND #perOn)) AND NOT #reset AND NOT #tempUpFlag;
   IF #_w1 THEN #statOut := #statOut - #tempStepWidth; END_IF;
   #tempDnFlag := #_w1;
END_REGION

REGION Network 10: standstill
   IF (#statDelta < #tempStepWidth) AND (#statDelta > #tempStepWidthNeg) AND NOT #reset AND #perOn AND NOT #tempUpFlag AND NOT #tempDnFlag THEN
       #statOut := #statInput;
   END_IF;
END_REGION

REGION Network 11: checking min. limit
   #statLow := (#statOut <= #realMin) AND NOT #reset;
   #lowLimit := #statLow;
END_REGION

REGION Network 12: min. limit reached
   IF NOT #reset AND #statLow THEN #statOut := #realMin; END_IF;
END_REGION

REGION Network 13: output and scaling to analog
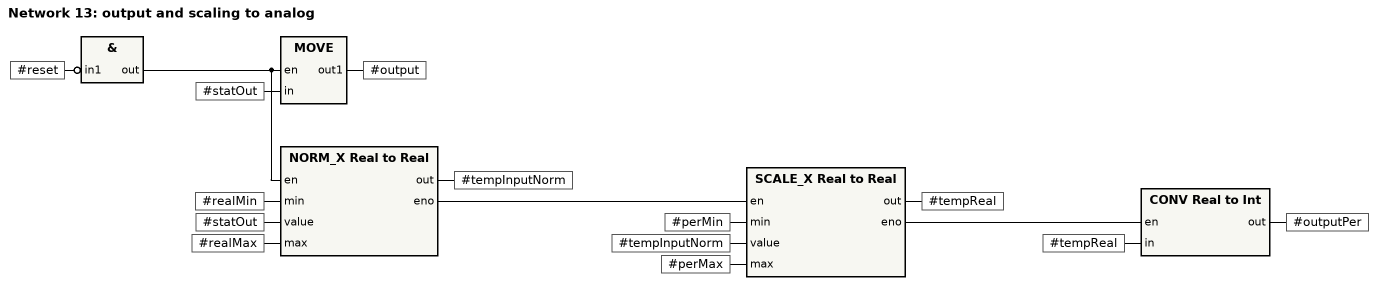
   // ENO of a box is taken as its EN; it also drops when the box reports an error
   IF NOT #reset THEN
       #output := #statOut;
       #tempInputNorm := NORM_X(MIN := #realMin, VALUE := #statOut, MAX := #realMax);
       #tempReal := SCALE_X(MIN := #perMin, VALUE := #tempInputNorm, MAX := #perMax);
       #outputPer := REAL_TO_INT(#tempReal);
   END_IF;
END_REGION
END_FUNCTION_BLOCK

ORGANIZATION_BLOCK "Level Indicating Controller 11"   // OB30, LAD, CyclicInterrupt
TITLE = Level Control Indicator
{ S7_Optimized_Access := 'TRUE' }
VERSION : 0.1
// Ladder and Block Program to Control Tanks Level Process
   VAR_INPUT
      Initial_Call : Bool;   // Initial call of this OB
      Event_Count : Int;   // Events discarded
   END_VAR
   VAR_TEMP   // added for the SCL form of the ladder/FBD networks
      _w1 : Bool;
   END_VAR
BEGIN

REGION Network 1: User Setpoint
   // User input their Setpoint for Level in Integer Percentage converted into Real Number for PID Setpoint (0-100)
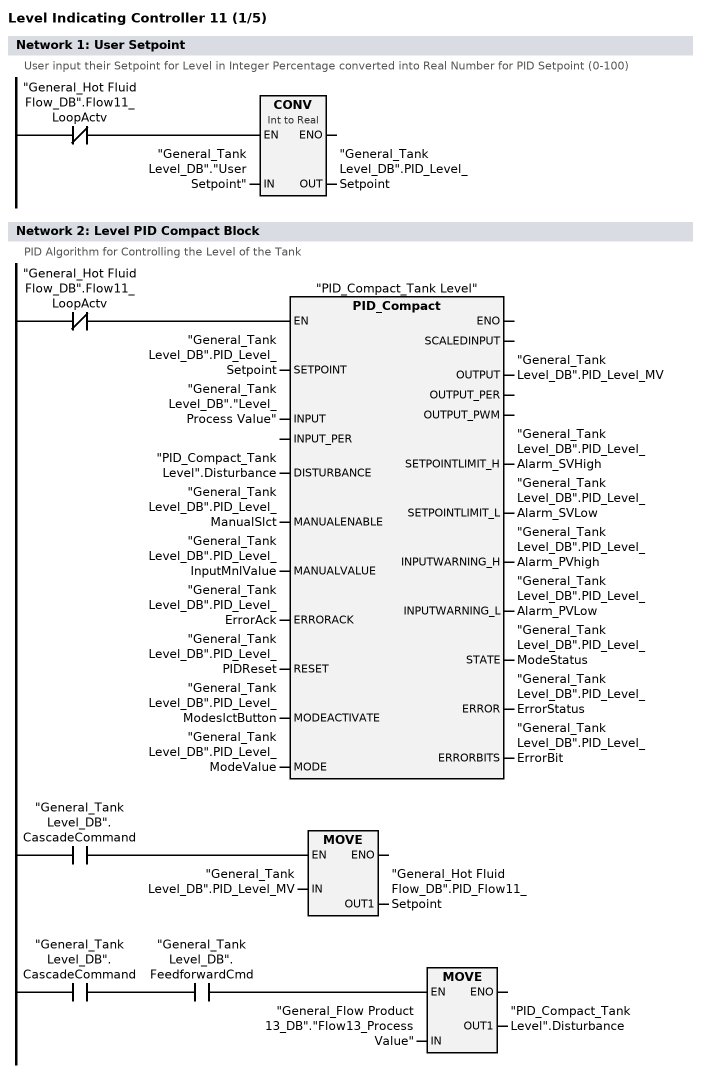
   RUNG wire#powerrail
      I_Contact( "General_Hot Fluid Flow_DB".Flow11_LoopActv )
      { S7_Templates := "[SrcType := Int, DestType := Real]" } Convert(in := "General_Tank Level_DB"."User Setpoint", out => "General_Tank Level_DB".PID_Level_Setpoint)
   END_RUNG
   // the same network as SCL:
   IF NOT "General_Hot Fluid Flow_DB".Flow11_LoopActv THEN
       "General_Tank Level_DB".PID_Level_Setpoint := INT_TO_REAL("General_Tank Level_DB"."User Setpoint");
   END_IF;
END_REGION

REGION Network 2: Level PID Compact Block
   // PID Algorithm for Controlling the Level of the Tank
   IF NOT "General_Hot Fluid Flow_DB".Flow11_LoopActv THEN
       "PID_Compact_Tank Level"(Setpoint := "General_Tank Level_DB".PID_Level_Setpoint,   // PID_Compact
                               Input := "General_Tank Level_DB"."Level_Process Value",
                               Disturbance := "PID_Compact_Tank Level".Disturbance,
                               ManualEnable := "General_Tank Level_DB".PID_Level_ManualSlct,
                               ManualValue := "General_Tank Level_DB".PID_Level_InputMnlValue,
                               ErrorAck := "General_Tank Level_DB".PID_Level_ErrorAck,
                               Reset := "General_Tank Level_DB".PID_Level_PIDReset,
                               ModeActivate := "General_Tank Level_DB".PID_Level_ModeslctButton,
                               Mode := "General_Tank Level_DB".PID_Level_ModeValue,
                               Output => "General_Tank Level_DB".PID_Level_MV,
                               SetpointLimit_H => "General_Tank Level_DB".PID_Level_Alarm_SVHigh,
                               SetpointLimit_L => "General_Tank Level_DB".PID_Level_Alarm_SVLow,
                               InputWarning_H => "General_Tank Level_DB".PID_Level_Alarm_PVhigh,
                               InputWarning_L => "General_Tank Level_DB".PID_Level_Alarm_PVLow,
                               State => "General_Tank Level_DB".PID_Level_ModeStatus,
                               Error => "General_Tank Level_DB".PID_Level_ErrorStatus,
                               ErrorBits => "General_Tank Level_DB".PID_Level_ErrorBit);
   END_IF;
   IF "General_Tank Level_DB".CascadeCommand THEN
       "General_Hot Fluid Flow_DB".PID_Flow11_Setpoint := "General_Tank Level_DB".PID_Level_MV;
   END_IF;
   IF "General_Tank Level_DB".CascadeCommand AND "General_Tank Level_DB".FeedforwardCmd THEN
       "PID_Compact_Tank Level".Disturbance := "General_Flow Product 13_DB"."Flow13_Process Value";
   END_IF;
END_REGION

REGION Network 3: Level Control Valve Control Block
   // Control Valve Process to Control the Tanks Level
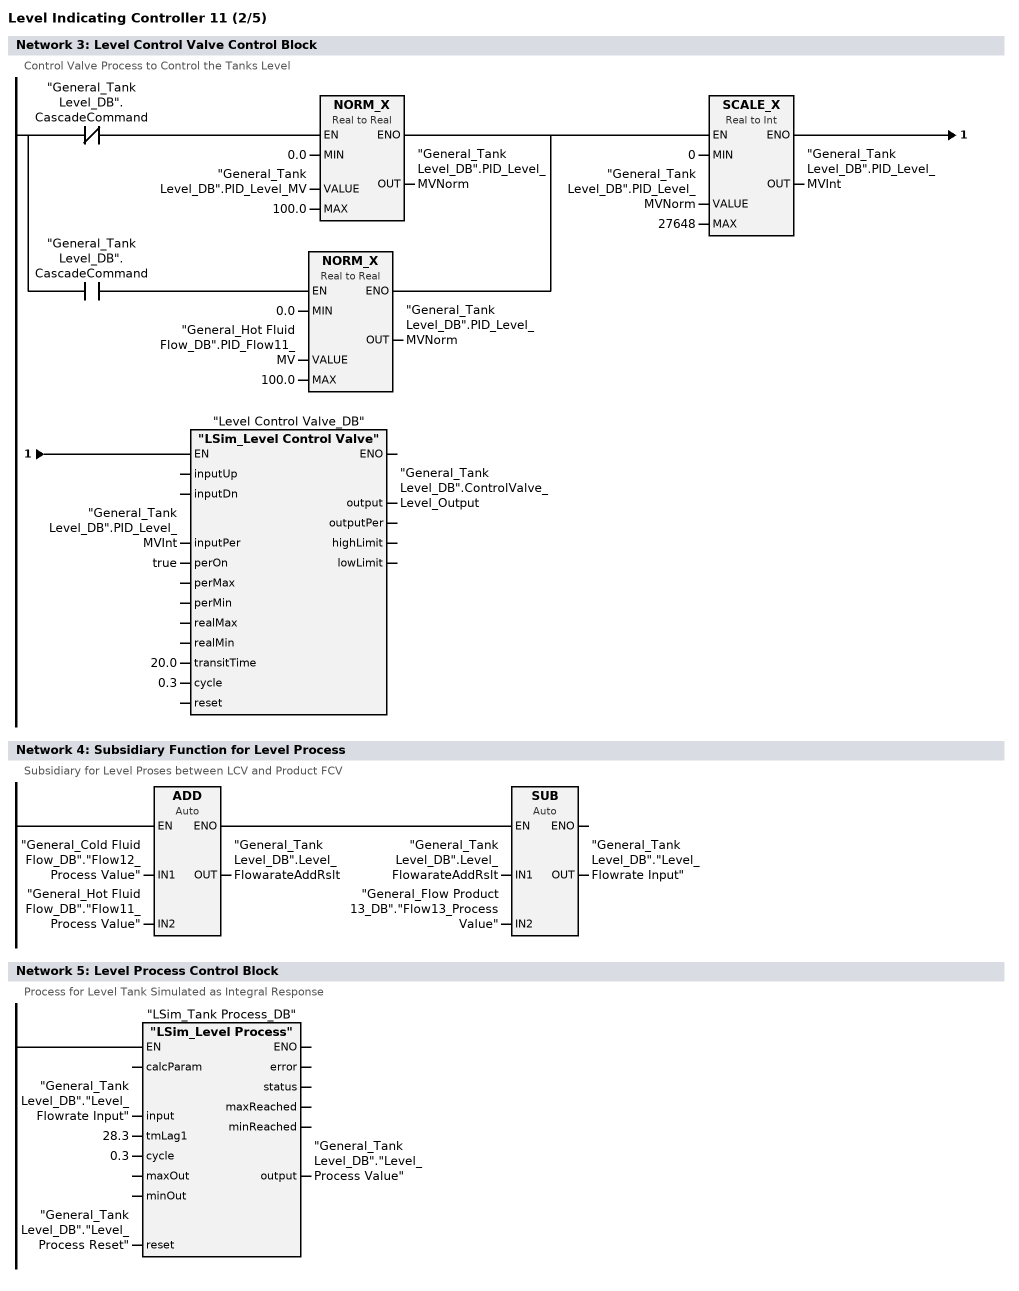
   RUNG wire#powerrail
      I_Contact( "General_Tank Level_DB".CascadeCommand )
      { S7_Templates := "[SrcType := Real, DestType := Real]" } Normalize(min := 0.0, value := "General_Tank Level_DB".PID_Level_MV, max := 100.0, out => "General_Tank Level_DB".PID_Level_MVNorm)
      wire#w1
      { S7_Templates := "[SrcType := Real, DestType := Int]" } Scale(min := 0, value := "General_Tank Level_DB".PID_Level_MVNorm, max := 27648, out => "General_Tank Level_DB".PID_Level_MVInt)
      "Level Control Valve_DB"(inputUp :=, inputDn :=, inputPer := "General_Tank Level_DB".PID_Level_MVInt, perOn := true, perMax :=, perMin :=, realMax :=, realMin :=, transitTime := 20.0, cycle := 0.3, reset :=, output => "General_Tank Level_DB".ControlValve_Level_Output, outputPer =>, highLimit =>, lowLimit =>)
   END_RUNG
   RUNG wire#powerrail
      Contact( "General_Tank Level_DB".CascadeCommand )
      { S7_Templates := "[SrcType := Real, DestType := Real]" } Normalize(min := 0.0, value := "General_Hot Fluid Flow_DB".PID_Flow11_MV, max := 100.0, out => "General_Tank Level_DB".PID_Level_MVNorm)
   END_RUNG wire#w1
   // the same network as SCL:
   #_w1 := NOT "General_Tank Level_DB".CascadeCommand;
   IF #_w1 THEN
       "General_Tank Level_DB".PID_Level_MVNorm := NORM_X(MIN := 0.0, VALUE := "General_Tank Level_DB".PID_Level_MV, MAX := 100.0);
   END_IF;
   IF "General_Tank Level_DB".CascadeCommand THEN
       "General_Tank Level_DB".PID_Level_MVNorm := NORM_X(MIN := 0.0, VALUE := "General_Hot Fluid Flow_DB".PID_Flow11_MV, MAX := 100.0);
   END_IF;
   IF #_w1 OR "General_Tank Level_DB".CascadeCommand THEN
       "General_Tank Level_DB".PID_Level_MVInt := SCALE_X(MIN := 0, VALUE := "General_Tank Level_DB".PID_Level_MVNorm, MAX := 27648);
       "Level Control Valve_DB"(inputPer := "General_Tank Level_DB".PID_Level_MVInt,   // "LSim_Level Control Valve"
                               perOn := true,
                               transitTime := 20.0,
                               cycle := 0.3,
                               output => "General_Tank Level_DB".ControlValve_Level_Output);
   END_IF;
END_REGION

REGION Network 4: Subsidiary Function for Level Process
   // Subsidiary for Level Proses between LCV and Product FCV
   RUNG wire#powerrail
      Add(in1 := "General_Cold Fluid Flow_DB"."Flow12_Process Value", in2 := "General_Hot Fluid Flow_DB"."Flow11_Process Value", out => "General_Tank Level_DB".Level_FlowarateAddRslt)
      Sub(in1 := "General_Tank Level_DB".Level_FlowarateAddRslt, in2 := "General_Flow Product 13_DB"."Flow13_Process Value", out => "General_Tank Level_DB"."Level_Flowrate Input")
   END_RUNG
   // the same network as SCL:
   "General_Tank Level_DB".Level_FlowarateAddRslt := "General_Cold Fluid Flow_DB"."Flow12_Process Value" + "General_Hot Fluid Flow_DB"."Flow11_Process Value";
   "General_Tank Level_DB"."Level_Flowrate Input" := "General_Tank Level_DB".Level_FlowarateAddRslt - "General_Flow Product 13_DB"."Flow13_Process Value";
END_REGION

REGION Network 5: Level Process Control Block
   // Process for Level Tank Simulated as Integral Response
   RUNG wire#powerrail
      "LSim_Tank Process_DB"(calcParam :=, input := "General_Tank Level_DB"."Level_Flowrate Input", tmLag1 := 28.3, cycle := 0.3, maxOut :=, minOut :=, reset := "General_Tank Level_DB"."Level_Process Reset", error =>, status =>, maxReached =>, minReached =>, output => "General_Tank Level_DB"."Level_Process Value")
   END_RUNG
   // the same network as SCL:
   "LSim_Tank Process_DB"(input := "General_Tank Level_DB"."Level_Flowrate Input",   // "LSim_Level Process"
                          tmLag1 := 28.3,
                          cycle := 0.3,
                          reset := "General_Tank Level_DB"."Level_Process Reset",
                          output => "General_Tank Level_DB"."Level_Process Value");
END_REGION

REGION Network 6: Safety Block For Level Limit
   // Set Alarm Limit for LSH and LSL activate when Level at 90% and 10%
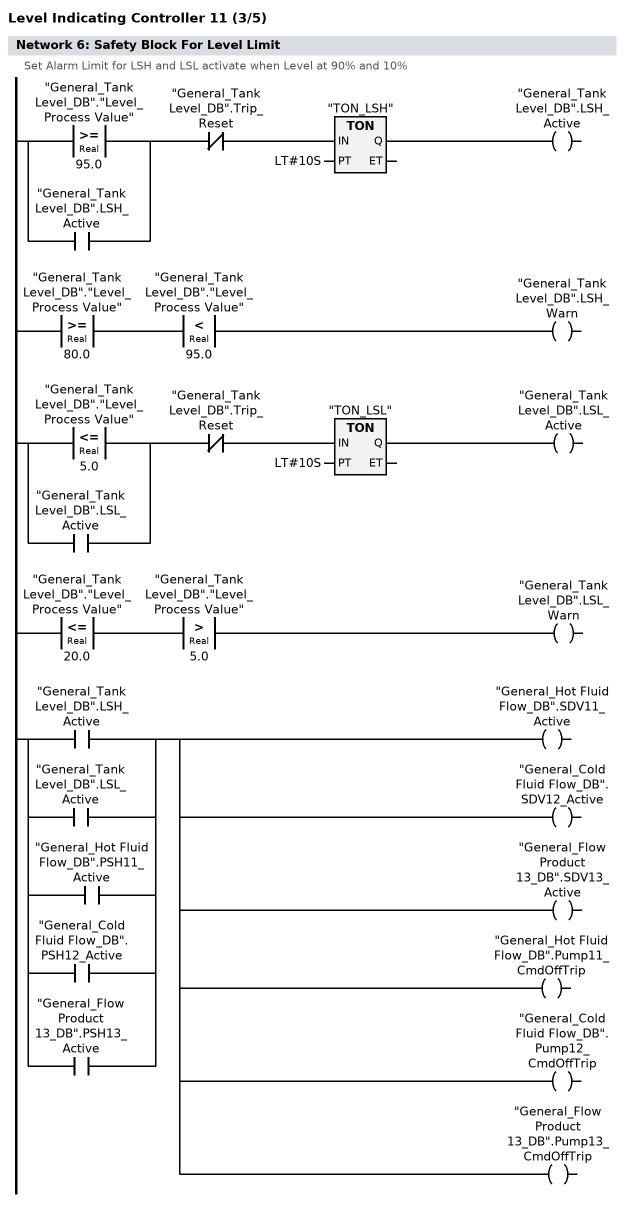
   "TON_LSH".TON(IN := (("General_Tank Level_DB"."Level_Process Value" >= 95.0) OR "General_Tank Level_DB".LSH_Active) AND NOT "General_Tank Level_DB".Trip_Reset,
                 PT := LT#10S);
   "General_Tank Level_DB".LSH_Active := "TON_LSH".Q;
   "General_Tank Level_DB".LSH_Warn := ("General_Tank Level_DB"."Level_Process Value" >= 80.0) AND ("General_Tank Level_DB"."Level_Process Value" < 95.0);
   "TON_LSL".TON(IN := (("General_Tank Level_DB"."Level_Process Value" <= 5.0) OR "General_Tank Level_DB".LSL_Active) AND NOT "General_Tank Level_DB".Trip_Reset,
                 PT := LT#10S);
   "General_Tank Level_DB".LSL_Active := "TON_LSL".Q;
   "General_Tank Level_DB".LSL_Warn := ("General_Tank Level_DB"."Level_Process Value" <= 20.0) AND ("General_Tank Level_DB"."Level_Process Value" > 5.0);
   "General_Hot Fluid Flow_DB".SDV11_Active := "General_Tank Level_DB".LSH_Active OR "General_Tank Level_DB".LSL_Active OR "General_Hot Fluid Flow_DB".PSH11_Active OR "General_Cold Fluid Flow_DB".PSH12_Active OR "General_Flow Product 13_DB".PSH13_Active;
   "General_Cold Fluid Flow_DB".SDV12_Active := "General_Hot Fluid Flow_DB".SDV11_Active;
   "General_Flow Product 13_DB".SDV13_Active := "General_Hot Fluid Flow_DB".SDV11_Active;
   "General_Hot Fluid Flow_DB".Pump11_CmdOffTrip := "General_Hot Fluid Flow_DB".SDV11_Active;
   "General_Cold Fluid Flow_DB".Pump12_CmdOffTrip := "General_Hot Fluid Flow_DB".SDV11_Active;
   "General_Flow Product 13_DB".Pump13_CmdOffTrip := "General_Hot Fluid Flow_DB".SDV11_Active;
END_REGION

REGION Network 7: Alarm Management Block
   // Control Block for Managing the Alarm Occured in the System
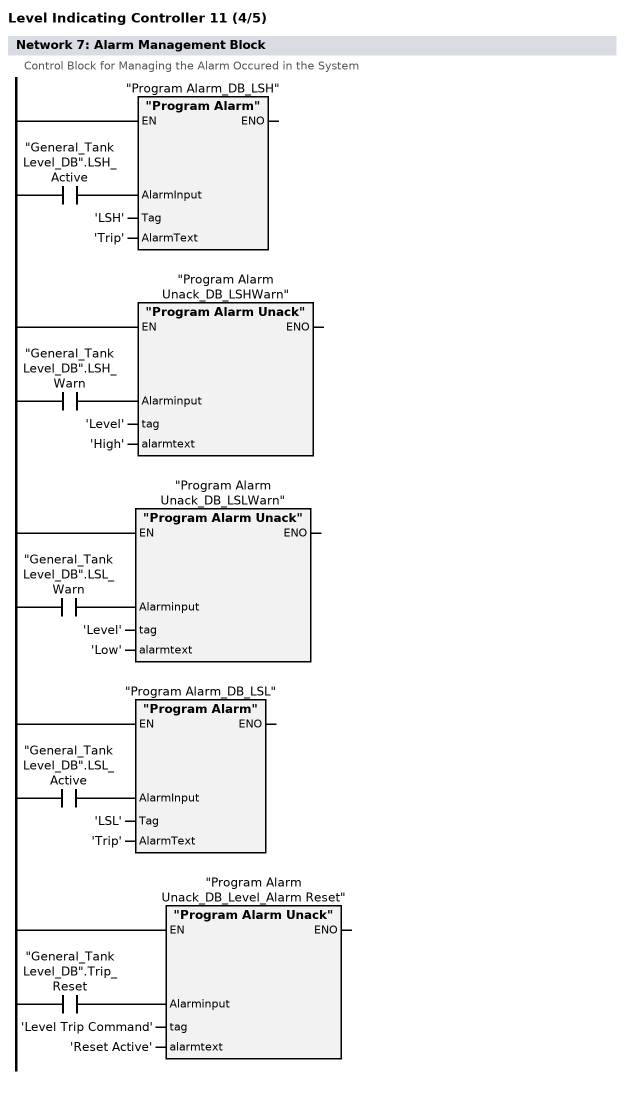
   RUNG wire#powerrail
      "Program Alarm_DB_LSH"(AlarmInput := wire#w1, Tag := 'LSH', AlarmText := 'Trip')
   END_RUNG
   RUNG wire#powerrail
      Contact( "General_Tank Level_DB".LSH_Active )
   END_RUNG wire#w1
   RUNG wire#powerrail
      "Program Alarm Unack_DB_LSHWarn"(Alarminput := wire#w2, tag := 'Level', alarmtext := 'High')
   END_RUNG
   RUNG wire#powerrail
      Contact( "General_Tank Level_DB".LSH_Warn )
   END_RUNG wire#w2
   RUNG wire#powerrail
      "Program Alarm Unack_DB_LSLWarn"(Alarminput := wire#w3, tag := 'Level', alarmtext := 'Low')
   END_RUNG
   RUNG wire#powerrail
      Contact( "General_Tank Level_DB".LSL_Warn )
   END_RUNG wire#w3
   RUNG wire#powerrail
      "Program Alarm_DB_LSL"(AlarmInput := wire#w4, Tag := 'LSL', AlarmText := 'Trip')
   END_RUNG
   RUNG wire#powerrail
      Contact( "General_Tank Level_DB".LSL_Active )
   END_RUNG wire#w4
   RUNG wire#powerrail
      "Program Alarm Unack_DB_Level_Alarm Reset"(Alarminput := wire#w5, tag := 'Level Trip Command', alarmtext := 'Reset Active')
   END_RUNG
   RUNG wire#powerrail
      Contact( "General_Tank Level_DB".Trip_Reset )
   END_RUNG wire#w5
   // the same network as SCL:
   "Program Alarm_DB_LSH"(AlarmInput := "General_Tank Level_DB".LSH_Active, Tag := 'LSH', AlarmText := 'Trip');   // "Program Alarm"
   "Program Alarm Unack_DB_LSHWarn"(Alarminput := "General_Tank Level_DB".LSH_Warn,   // "Program Alarm Unack"
                           tag := 'Level',
                           alarmtext := 'High');
   "Program Alarm Unack_DB_LSLWarn"(Alarminput := "General_Tank Level_DB".LSL_Warn,   // "Program Alarm Unack"
                           tag := 'Level',
                           alarmtext := 'Low');
   "Program Alarm_DB_LSL"(AlarmInput := "General_Tank Level_DB".LSL_Active, Tag := 'LSL', AlarmText := 'Trip');   // "Program Alarm"
   "Program Alarm Unack_DB_Level_Alarm Reset"(Alarminput := "General_Tank Level_DB".Trip_Reset,   // "Program Alarm Unack"
                           tag := 'Level Trip Command',
                           alarmtext := 'Reset Active');
END_REGION

REGION Network 8: User Additional Feature
   // Put additional feature that user can use to easier the system operation
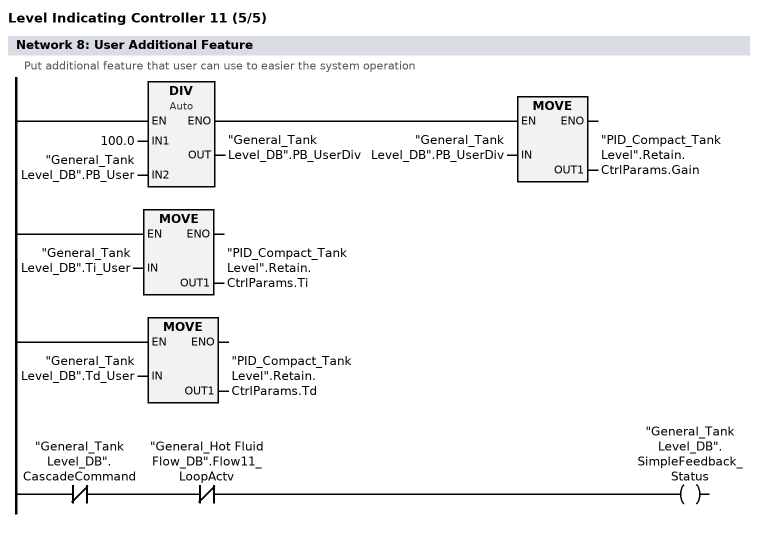
   RUNG wire#powerrail
      Div(in1 := 100.0, in2 := "General_Tank Level_DB".PB_User, out => "General_Tank Level_DB".PB_UserDiv)
      Move(in := "General_Tank Level_DB".PB_UserDiv, out1 => "PID_Compact_Tank Level".Retain.CtrlParams.Gain)
   END_RUNG
   RUNG wire#powerrail
      Move(in := "General_Tank Level_DB".Ti_User, out1 => "PID_Compact_Tank Level".Retain.CtrlParams.Ti)
   END_RUNG
   RUNG wire#powerrail
      Move(in := "General_Tank Level_DB".Td_User, out1 => "PID_Compact_Tank Level".Retain.CtrlParams.Td)
   END_RUNG
   RUNG wire#powerrail
      I_Contact( "General_Tank Level_DB".CascadeCommand )
      I_Contact( "General_Hot Fluid Flow_DB".Flow11_LoopActv )
      Coil( "General_Tank Level_DB".SimpleFeedback_Status )
   END_RUNG
   // the same network as SCL:
   "General_Tank Level_DB".PB_UserDiv := 100.0 / "General_Tank Level_DB".PB_User;
   "PID_Compact_Tank Level".Retain.CtrlParams.Gain := "General_Tank Level_DB".PB_UserDiv;
   "PID_Compact_Tank Level".Retain.CtrlParams.Ti := "General_Tank Level_DB".Ti_User;
   "PID_Compact_Tank Level".Retain.CtrlParams.Td := "General_Tank Level_DB".Td_User;
   "General_Tank Level_DB".SimpleFeedback_Status := NOT "General_Tank Level_DB".CascadeCommand AND NOT "General_Hot Fluid Flow_DB".Flow11_LoopActv;
END_REGION
END_ORGANIZATION_BLOCK

ORGANIZATION_BLOCK "Flow Indicating Controller 13"   // OB31, LAD, CyclicInterrupt
TITLE = Flow Indicator Controller 13 (Product)
{ S7_Optimized_Access := 'TRUE' }
VERSION : 0.1
// Ladder and Block Program to control flowrate of Product (Tank Output)
   VAR_INPUT
      Initial_Call : Bool;   // Initial call of this OB
      Event_Count : Int;   // Events discarded
   END_VAR
BEGIN

REGION Network 1: User Setpoint
   // User input their Setpoint for flowrate in L/s  converted into Real Number for PID Setpoint (0-100)
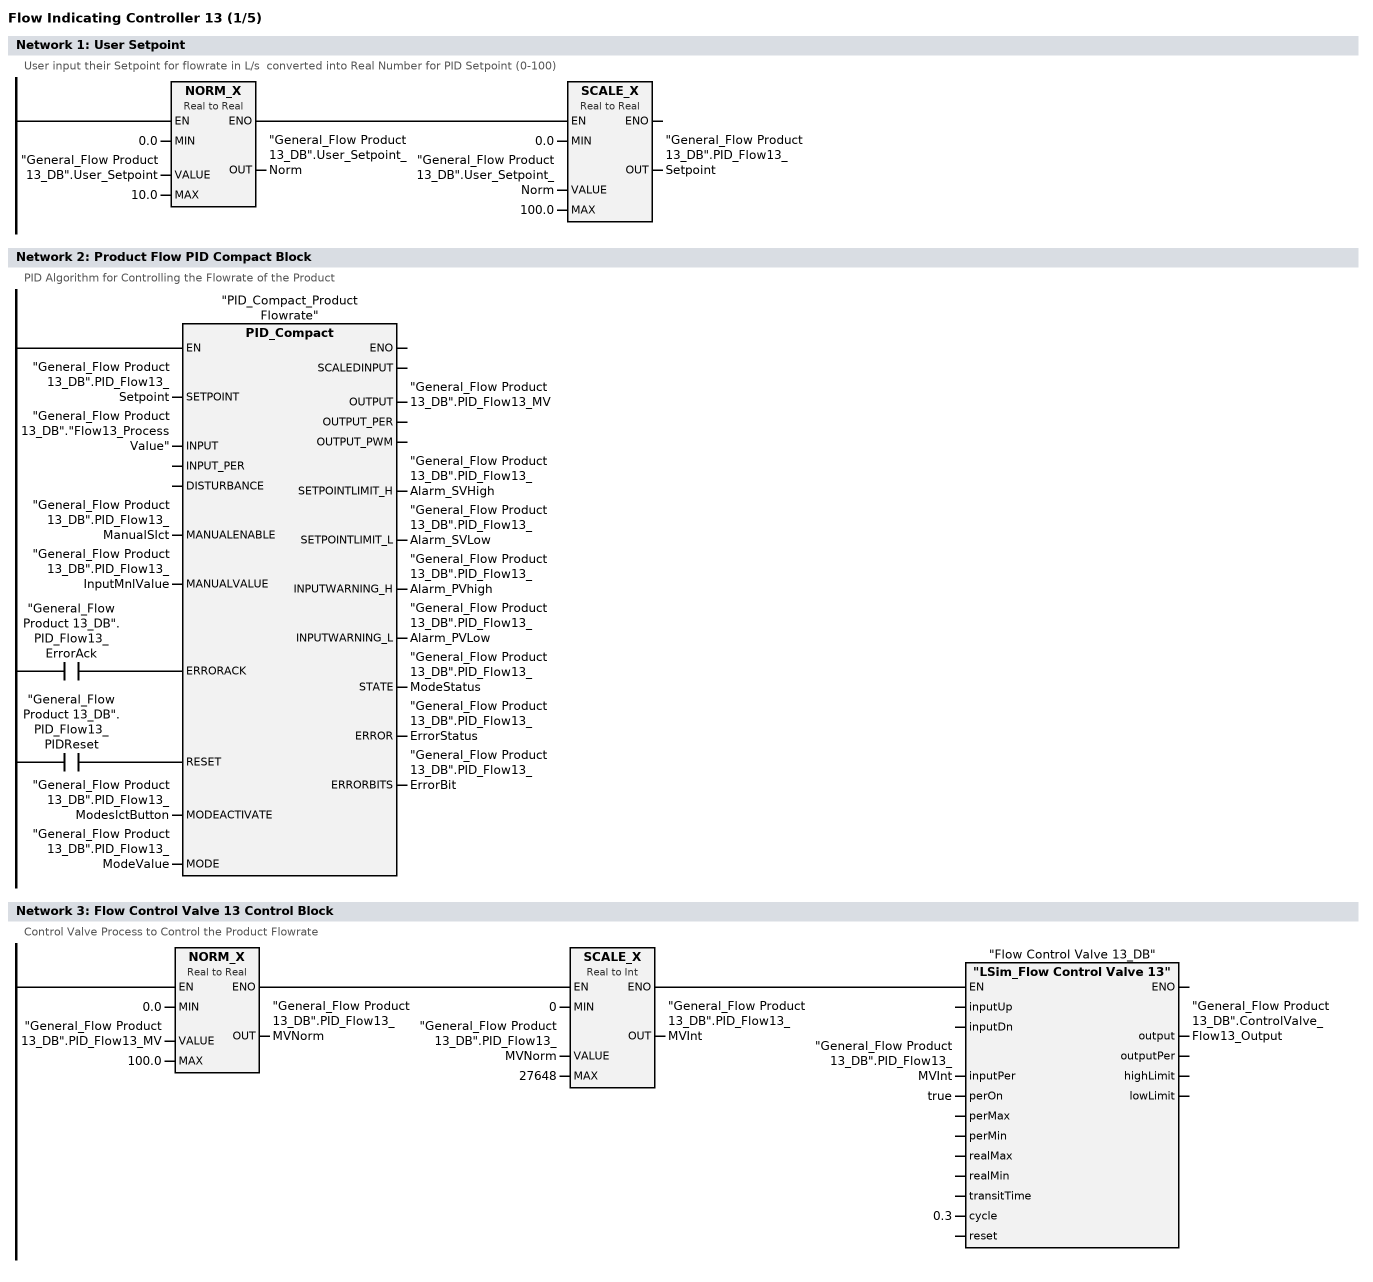
   RUNG wire#powerrail
      { S7_Templates := "[SrcType := Real, DestType := Real]" } Normalize(min := 0.0, value := "General_Flow Product 13_DB".User_Setpoint, max := 10.0, out => "General_Flow Product 13_DB".User_Setpoint_Norm)
      { S7_Templates := "[SrcType := Real, DestType := Real]" } Scale(min := 0.0, value := "General_Flow Product 13_DB".User_Setpoint_Norm, max := 100.0, out => "General_Flow Product 13_DB".PID_Flow13_Setpoint)
   END_RUNG
   // the same network as SCL:
   "General_Flow Product 13_DB".User_Setpoint_Norm := NORM_X(MIN := 0.0, VALUE := "General_Flow Product 13_DB".User_Setpoint, MAX := 10.0);
   "General_Flow Product 13_DB".PID_Flow13_Setpoint := SCALE_X(MIN := 0.0, VALUE := "General_Flow Product 13_DB".User_Setpoint_Norm, MAX := 100.0);
END_REGION

REGION Network 2: Product Flow PID Compact Block
   // PID Algorithm for Controlling the Flowrate of the Product
   "PID_Compact_Product Flowrate"(Setpoint := "General_Flow Product 13_DB".PID_Flow13_Setpoint,   // PID_Compact
                           Input := "General_Flow Product 13_DB"."Flow13_Process Value",
                           ManualEnable := "General_Flow Product 13_DB".PID_Flow13_ManualSlct,
                           ManualValue := "General_Flow Product 13_DB".PID_Flow13_InputMnlValue,
                           ErrorAck := "General_Flow Product 13_DB".PID_Flow13_ErrorAck,
                           Reset := "General_Flow Product 13_DB".PID_Flow13_PIDReset,
                           ModeActivate := "General_Flow Product 13_DB".PID_Flow13_ModeslctButton,
                           Mode := "General_Flow Product 13_DB".PID_Flow13_ModeValue,
                           Output => "General_Flow Product 13_DB".PID_Flow13_MV,
                           SetpointLimit_H => "General_Flow Product 13_DB".PID_Flow13_Alarm_SVHigh,
                           SetpointLimit_L => "General_Flow Product 13_DB".PID_Flow13_Alarm_SVLow,
                           InputWarning_H => "General_Flow Product 13_DB".PID_Flow13_Alarm_PVhigh,
                           InputWarning_L => "General_Flow Product 13_DB".PID_Flow13_Alarm_PVLow,
                           State => "General_Flow Product 13_DB".PID_Flow13_ModeStatus,
                           Error => "General_Flow Product 13_DB".PID_Flow13_ErrorStatus,
                           ErrorBits => "General_Flow Product 13_DB".PID_Flow13_ErrorBit);
END_REGION

REGION Network 3: Flow Control Valve 13 Control Block
   // Control Valve Process to Control the Product Flowrate
   RUNG wire#powerrail
      { S7_Templates := "[SrcType := Real, DestType := Real]" } Normalize(min := 0.0, value := "General_Flow Product 13_DB".PID_Flow13_MV, max := 100.0, out => "General_Flow Product 13_DB".PID_Flow13_MVNorm)
      { S7_Templates := "[SrcType := Real, DestType := Int]" } Scale(min := 0, value := "General_Flow Product 13_DB".PID_Flow13_MVNorm, max := 27648, out => "General_Flow Product 13_DB".PID_Flow13_MVInt)
      "Flow Control Valve 13_DB"(inputUp :=, inputDn :=, inputPer := "General_Flow Product 13_DB".PID_Flow13_MVInt, perOn := true, perMax :=, perMin :=, realMax :=, realMin :=, transitTime :=, cycle := 0.3, reset :=, output => "General_Flow Product 13_DB".ControlValve_Flow13_Output, outputPer =>, highLimit =>, lowLimit =>)
   END_RUNG
   // the same network as SCL:
   "General_Flow Product 13_DB".PID_Flow13_MVNorm := NORM_X(MIN := 0.0, VALUE := "General_Flow Product 13_DB".PID_Flow13_MV, MAX := 100.0);
   "General_Flow Product 13_DB".PID_Flow13_MVInt := SCALE_X(MIN := 0, VALUE := "General_Flow Product 13_DB".PID_Flow13_MVNorm, MAX := 27648);
   "Flow Control Valve 13_DB"(inputPer := "General_Flow Product 13_DB".PID_Flow13_MVInt,   // "LSim_Flow Control Valve 13"
                           perOn := true,
                           cycle := 0.3,
                           output => "General_Flow Product 13_DB".ControlValve_Flow13_Output);
END_REGION

REGION Network 4: Product Flow 13 Process Control Block
   // Process for Flowrate as First Order System
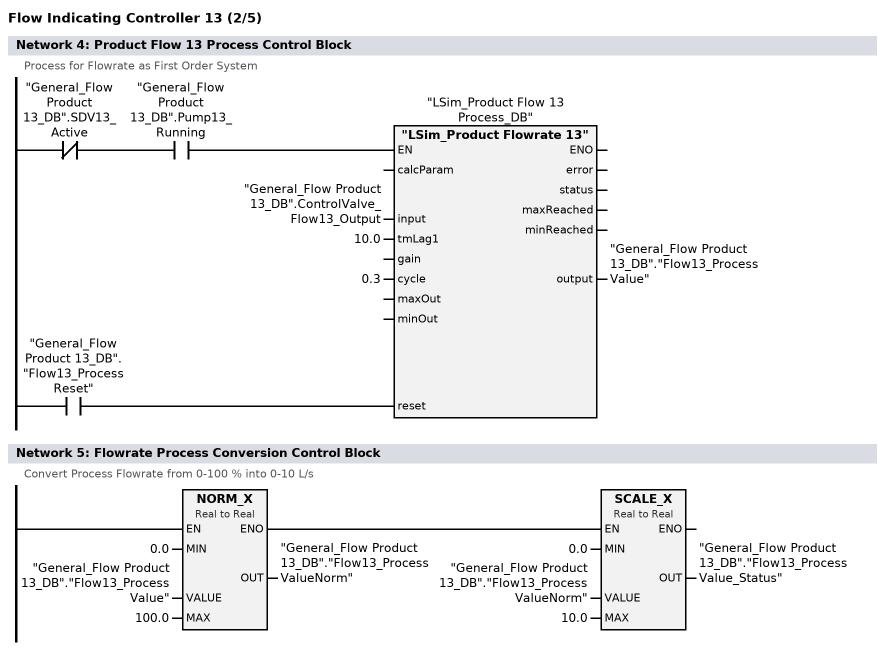
   RUNG wire#powerrail
      I_Contact( "General_Flow Product 13_DB".SDV13_Active )
      Contact( "General_Flow Product 13_DB".Pump13_Running )
      "LSim_Product Flow 13 Process_DB"(reset := wire#w1, calcParam :=, input := "General_Flow Product 13_DB".ControlValve_Flow13_Output, tmLag1 := 10.0, gain :=, cycle := 0.3, maxOut :=, minOut :=, error =>, status =>, maxReached =>, minReached =>, output => "General_Flow Product 13_DB"."Flow13_Process Value")
   END_RUNG
   RUNG wire#powerrail
      Contact( "General_Flow Product 13_DB"."Flow13_Process Reset" )
   END_RUNG wire#w1
   // the same network as SCL:
   IF NOT "General_Flow Product 13_DB".SDV13_Active AND "General_Flow Product 13_DB".Pump13_Running THEN
       "LSim_Product Flow 13 Process_DB"(input := "General_Flow Product 13_DB".ControlValve_Flow13_Output,   // "LSim_Product Flowrate 13"
                               tmLag1 := 10.0,
                               cycle := 0.3,
                               reset := "General_Flow Product 13_DB"."Flow13_Process Reset",
                               output => "General_Flow Product 13_DB"."Flow13_Process Value");
   END_IF;
END_REGION

REGION Network 5: Flowrate Process Conversion Control Block
   // Convert Process Flowrate from 0-100 % into 0-10 L/s
   RUNG wire#powerrail
      { S7_Templates := "[SrcType := Real, DestType := Real]" } Normalize(min := 0.0, value := "General_Flow Product 13_DB"."Flow13_Process Value", max := 100.0, out => "General_Flow Product 13_DB"."Flow13_Process ValueNorm")
      { S7_Templates := "[SrcType := Real, DestType := Real]" } Scale(min := 0.0, value := "General_Flow Product 13_DB"."Flow13_Process ValueNorm", max := 10.0, out => "General_Flow Product 13_DB"."Flow13_Process Value_Status")
   END_RUNG
   // the same network as SCL:
   "General_Flow Product 13_DB"."Flow13_Process ValueNorm" := NORM_X(MIN := 0.0, VALUE := "General_Flow Product 13_DB"."Flow13_Process Value", MAX := 100.0);
   "General_Flow Product 13_DB"."Flow13_Process Value_Status" := SCALE_X(MIN := 0.0, VALUE := "General_Flow Product 13_DB"."Flow13_Process ValueNorm", MAX := 10.0);
END_REGION

REGION Network 6: Pump Operational Control Block
   // Block for Controlling On/Off of the Pump and It's Safety Operation
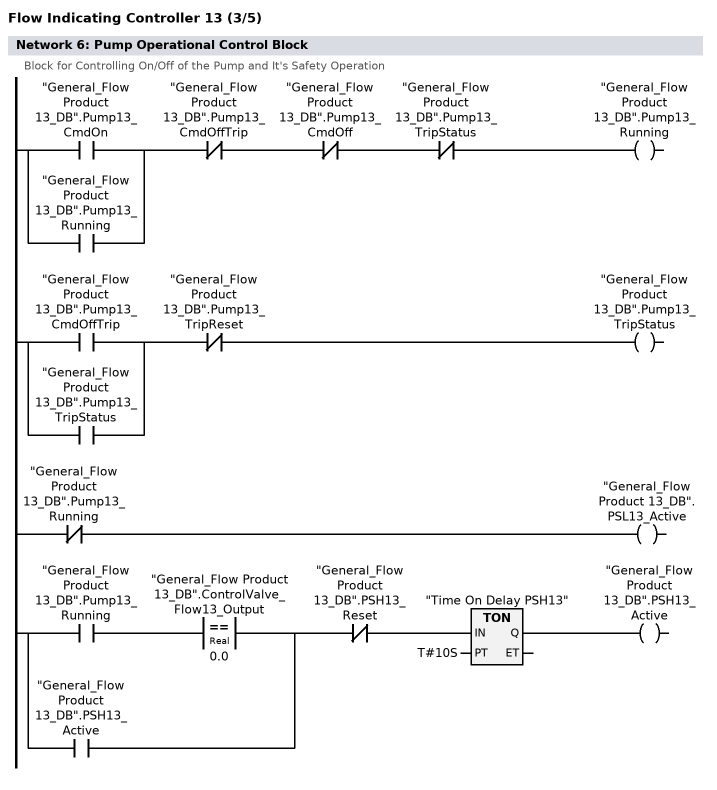
   "General_Flow Product 13_DB".Pump13_Running := ("General_Flow Product 13_DB".Pump13_CmdOn OR "General_Flow Product 13_DB".Pump13_Running) AND NOT "General_Flow Product 13_DB".Pump13_CmdOffTrip AND NOT "General_Flow Product 13_DB".Pump13_CmdOff AND NOT "General_Flow Product 13_DB".Pump13_TripStatus;
   "General_Flow Product 13_DB".Pump13_TripStatus := ("General_Flow Product 13_DB".Pump13_CmdOffTrip OR "General_Flow Product 13_DB".Pump13_TripStatus) AND NOT "General_Flow Product 13_DB".Pump13_TripReset;
   "General_Flow Product 13_DB".PSL13_Active := NOT "General_Flow Product 13_DB".Pump13_Running;
   "Time On Delay PSH13".TON(IN := (("General_Flow Product 13_DB".Pump13_Running AND ("General_Flow Product 13_DB".ControlValve_Flow13_Output = 0.0)) OR "General_Flow Product 13_DB".PSH13_Active) AND NOT "General_Flow Product 13_DB".PSH13_Reset,
                           PT := T#10S);
   "General_Flow Product 13_DB".PSH13_Active := "Time On Delay PSH13".Q;
END_REGION

REGION Network 7: Alarm Management Block
   // Control Block for Managing the Alarm Occured in the System
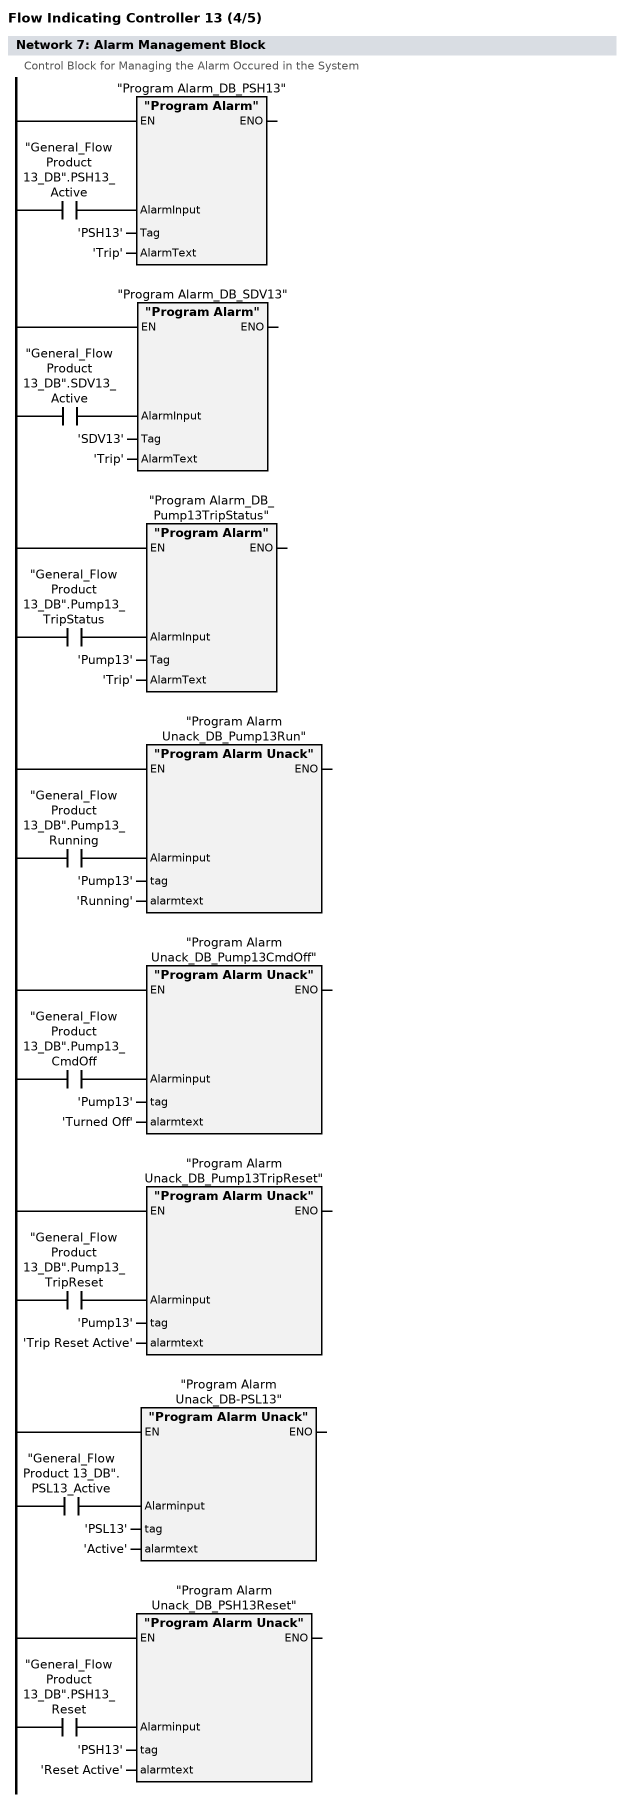
   RUNG wire#powerrail
      "Program Alarm_DB_PSH13"(AlarmInput := wire#w1, Tag := 'PSH13', AlarmText := 'Trip')
   END_RUNG
   RUNG wire#powerrail
      Contact( "General_Flow Product 13_DB".PSH13_Active )
   END_RUNG wire#w1
   RUNG wire#powerrail
      "Program Alarm_DB_SDV13"(AlarmInput := wire#w2, Tag := 'SDV13', AlarmText := 'Trip')
   END_RUNG
   RUNG wire#powerrail
      Contact( "General_Flow Product 13_DB".SDV13_Active )
   END_RUNG wire#w2
   RUNG wire#powerrail
      "Program Alarm_DB_Pump13TripStatus"(AlarmInput := wire#w3, Tag := 'Pump13', AlarmText := 'Trip')
   END_RUNG
   RUNG wire#powerrail
      Contact( "General_Flow Product 13_DB".Pump13_TripStatus )
   END_RUNG wire#w3
   RUNG wire#powerrail
      "Program Alarm Unack_DB_Pump13Run"(Alarminput := wire#w4, tag := 'Pump13', alarmtext := 'Running')
   END_RUNG
   RUNG wire#powerrail
      Contact( "General_Flow Product 13_DB".Pump13_Running )
   END_RUNG wire#w4
   RUNG wire#powerrail
      "Program Alarm Unack_DB_Pump13CmdOff"(Alarminput := wire#w5, tag := 'Pump13', alarmtext := 'Turned Off')
   END_RUNG
   RUNG wire#powerrail
      Contact( "General_Flow Product 13_DB".Pump13_CmdOff )
   END_RUNG wire#w5
   RUNG wire#powerrail
      "Program Alarm Unack_DB_Pump13TripReset"(Alarminput := wire#w6, tag := 'Pump13', alarmtext := 'Trip Reset Active')
   END_RUNG
   RUNG wire#powerrail
      Contact( "General_Flow Product 13_DB".Pump13_TripReset )
   END_RUNG wire#w6
   RUNG wire#powerrail
      "Program Alarm Unack_DB-PSL13"(Alarminput := wire#w7, tag := 'PSL13', alarmtext := 'Active')
   END_RUNG
   RUNG wire#powerrail
      Contact( "General_Flow Product 13_DB".PSL13_Active )
   END_RUNG wire#w7
   RUNG wire#powerrail
      "Program Alarm Unack_DB_PSH13Reset"(Alarminput := wire#w8, tag := 'PSH13', alarmtext := 'Reset Active')
   END_RUNG
   RUNG wire#powerrail
      Contact( "General_Flow Product 13_DB".PSH13_Reset )
   END_RUNG wire#w8
   // the same network as SCL:
   "Program Alarm_DB_PSH13"(AlarmInput := "General_Flow Product 13_DB".PSH13_Active,   // "Program Alarm"
                           Tag := 'PSH13',
                           AlarmText := 'Trip');
   "Program Alarm_DB_SDV13"(AlarmInput := "General_Flow Product 13_DB".SDV13_Active,   // "Program Alarm"
                           Tag := 'SDV13',
                           AlarmText := 'Trip');
   "Program Alarm_DB_Pump13TripStatus"(AlarmInput := "General_Flow Product 13_DB".Pump13_TripStatus,   // "Program Alarm"
                           Tag := 'Pump13',
                           AlarmText := 'Trip');
   "Program Alarm Unack_DB_Pump13Run"(Alarminput := "General_Flow Product 13_DB".Pump13_Running,   // "Program Alarm Unack"
                           tag := 'Pump13',
                           alarmtext := 'Running');
   "Program Alarm Unack_DB_Pump13CmdOff"(Alarminput := "General_Flow Product 13_DB".Pump13_CmdOff,   // "Program Alarm Unack"
                           tag := 'Pump13',
                           alarmtext := 'Turned Off');
   "Program Alarm Unack_DB_Pump13TripReset"(Alarminput := "General_Flow Product 13_DB".Pump13_TripReset,   // "Program Alarm Unack"
                           tag := 'Pump13',
                           alarmtext := 'Trip Reset Active');
   "Program Alarm Unack_DB-PSL13"(Alarminput := "General_Flow Product 13_DB".PSL13_Active,   // "Program Alarm Unack"
                           tag := 'PSL13',
                           alarmtext := 'Active');
   "Program Alarm Unack_DB_PSH13Reset"(Alarminput := "General_Flow Product 13_DB".PSH13_Reset,   // "Program Alarm Unack"
                           tag := 'PSH13',
                           alarmtext := 'Reset Active');
END_REGION

REGION Network 8: User Additional Feature
   // Put additional feature that user can use to easier the system operation
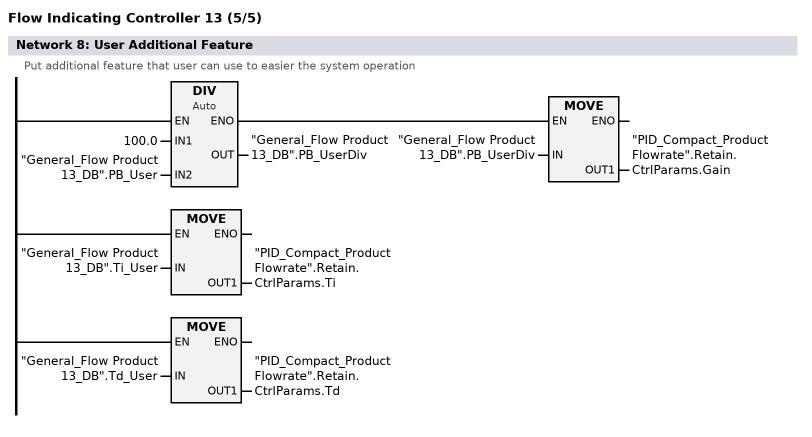
   RUNG wire#powerrail
      Div(in1 := 100.0, in2 := "General_Flow Product 13_DB".PB_User, out => "General_Flow Product 13_DB".PB_UserDiv)
      Move(in := "General_Flow Product 13_DB".PB_UserDiv, out1 => "PID_Compact_Product Flowrate".Retain.CtrlParams.Gain)
   END_RUNG
   RUNG wire#powerrail
      Move(in := "General_Flow Product 13_DB".Ti_User, out1 => "PID_Compact_Product Flowrate".Retain.CtrlParams.Ti)
   END_RUNG
   RUNG wire#powerrail
      Move(in := "General_Flow Product 13_DB".Td_User, out1 => "PID_Compact_Product Flowrate".Retain.CtrlParams.Td)
   END_RUNG
   // the same network as SCL:
   "General_Flow Product 13_DB".PB_UserDiv := 100.0 / "General_Flow Product 13_DB".PB_User;
   "PID_Compact_Product Flowrate".Retain.CtrlParams.Gain := "General_Flow Product 13_DB".PB_UserDiv;
   "PID_Compact_Product Flowrate".Retain.CtrlParams.Ti := "General_Flow Product 13_DB".Ti_User;
   "PID_Compact_Product Flowrate".Retain.CtrlParams.Td := "General_Flow Product 13_DB".Td_User;
END_REGION
END_ORGANIZATION_BLOCK

ORGANIZATION_BLOCK "Temperature Indicating Controller"   // OB32, LAD, CyclicInterrupt
TITLE = Temperature Control Indicator
{ S7_Optimized_Access := 'TRUE' }
VERSION : 0.1
// Ladder and Block Program to Control Products Temperature
   VAR_INPUT
      Initial_Call : Bool;   // Initial call of this OB
      Event_Count : Int;   // Events discarded
   END_VAR
BEGIN

REGION Network 1: User Setpoint
   // User input their Setpoint for Temperature in Integer Percentage converted into Real Number for PID Setpoint (0-100)
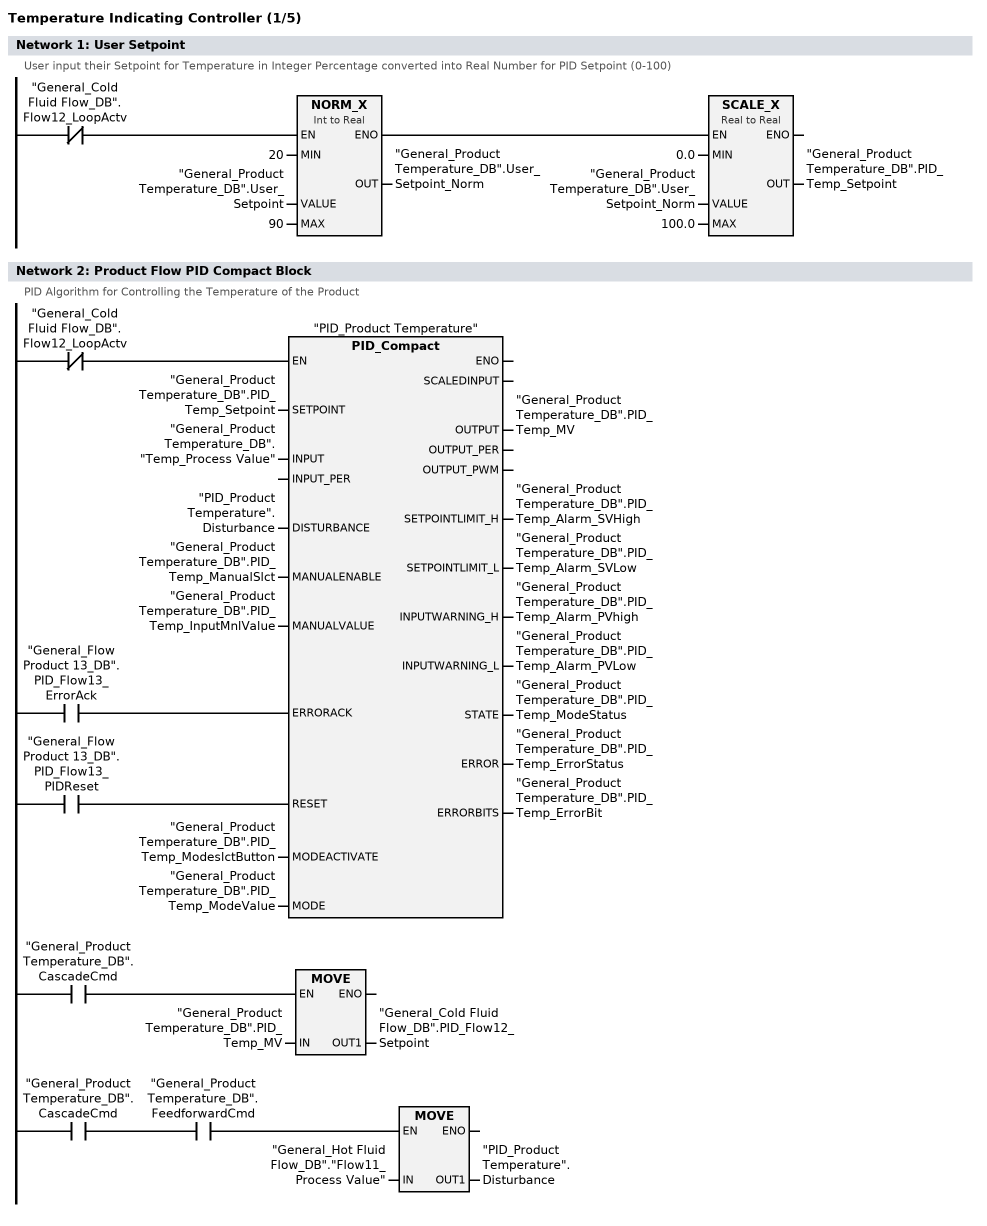
   RUNG wire#powerrail
      I_Contact( "General_Cold Fluid Flow_DB".Flow12_LoopActv )
      { S7_Templates := "[SrcType := Int, DestType := Real]" } Normalize(min := 20, value := "General_Product Temperature_DB".User_Setpoint, max := 90, out => "General_Product Temperature_DB".User_Setpoint_Norm)
      { S7_Templates := "[SrcType := Real, DestType := Real]" } Scale(min := 0.0, value := "General_Product Temperature_DB".User_Setpoint_Norm, max := 100.0, out => "General_Product Temperature_DB".PID_Temp_Setpoint)
   END_RUNG
   // the same network as SCL:
   IF NOT "General_Cold Fluid Flow_DB".Flow12_LoopActv THEN
       "General_Product Temperature_DB".User_Setpoint_Norm := NORM_X(MIN := 20, VALUE := "General_Product Temperature_DB".User_Setpoint, MAX := 90);
       "General_Product Temperature_DB".PID_Temp_Setpoint := SCALE_X(MIN := 0.0, VALUE := "General_Product Temperature_DB".User_Setpoint_Norm, MAX := 100.0);
   END_IF;
END_REGION

REGION Network 2: Product Flow PID Compact Block
   // PID Algorithm for Controlling the Temperature of the Product
   IF NOT "General_Cold Fluid Flow_DB".Flow12_LoopActv THEN
       "PID_Product Temperature"(Setpoint := "General_Product Temperature_DB".PID_Temp_Setpoint,   // PID_Compact
                               Input := "General_Product Temperature_DB"."Temp_Process Value",
                               Disturbance := "PID_Product Temperature".Disturbance,
                               ManualEnable := "General_Product Temperature_DB".PID_Temp_ManualSlct,
                               ManualValue := "General_Product Temperature_DB".PID_Temp_InputMnlValue,
                               ErrorAck := "General_Flow Product 13_DB".PID_Flow13_ErrorAck,
                               Reset := "General_Flow Product 13_DB".PID_Flow13_PIDReset,
                               ModeActivate := "General_Product Temperature_DB".PID_Temp_ModeslctButton,
                               Mode := "General_Product Temperature_DB".PID_Temp_ModeValue,
                               Output => "General_Product Temperature_DB".PID_Temp_MV,
                               SetpointLimit_H => "General_Product Temperature_DB".PID_Temp_Alarm_SVHigh,
                               SetpointLimit_L => "General_Product Temperature_DB".PID_Temp_Alarm_SVLow,
                               InputWarning_H => "General_Product Temperature_DB".PID_Temp_Alarm_PVhigh,
                               InputWarning_L => "General_Product Temperature_DB".PID_Temp_Alarm_PVLow,
                               State => "General_Product Temperature_DB".PID_Temp_ModeStatus,
                               Error => "General_Product Temperature_DB".PID_Temp_ErrorStatus,
                               ErrorBits => "General_Product Temperature_DB".PID_Temp_ErrorBit);
   END_IF;
   IF "General_Product Temperature_DB".CascadeCmd THEN
       "General_Cold Fluid Flow_DB".PID_Flow12_Setpoint := "General_Product Temperature_DB".PID_Temp_MV;
   END_IF;
   IF "General_Product Temperature_DB".CascadeCmd AND "General_Product Temperature_DB".FeedforwardCmd THEN
       "PID_Product Temperature".Disturbance := "General_Hot Fluid Flow_DB"."Flow11_Process Value";
   END_IF;
END_REGION

REGION Network 3: Temperature Control Valve 13 Control Block
   // Control Valve Process to Control the Product Temperature
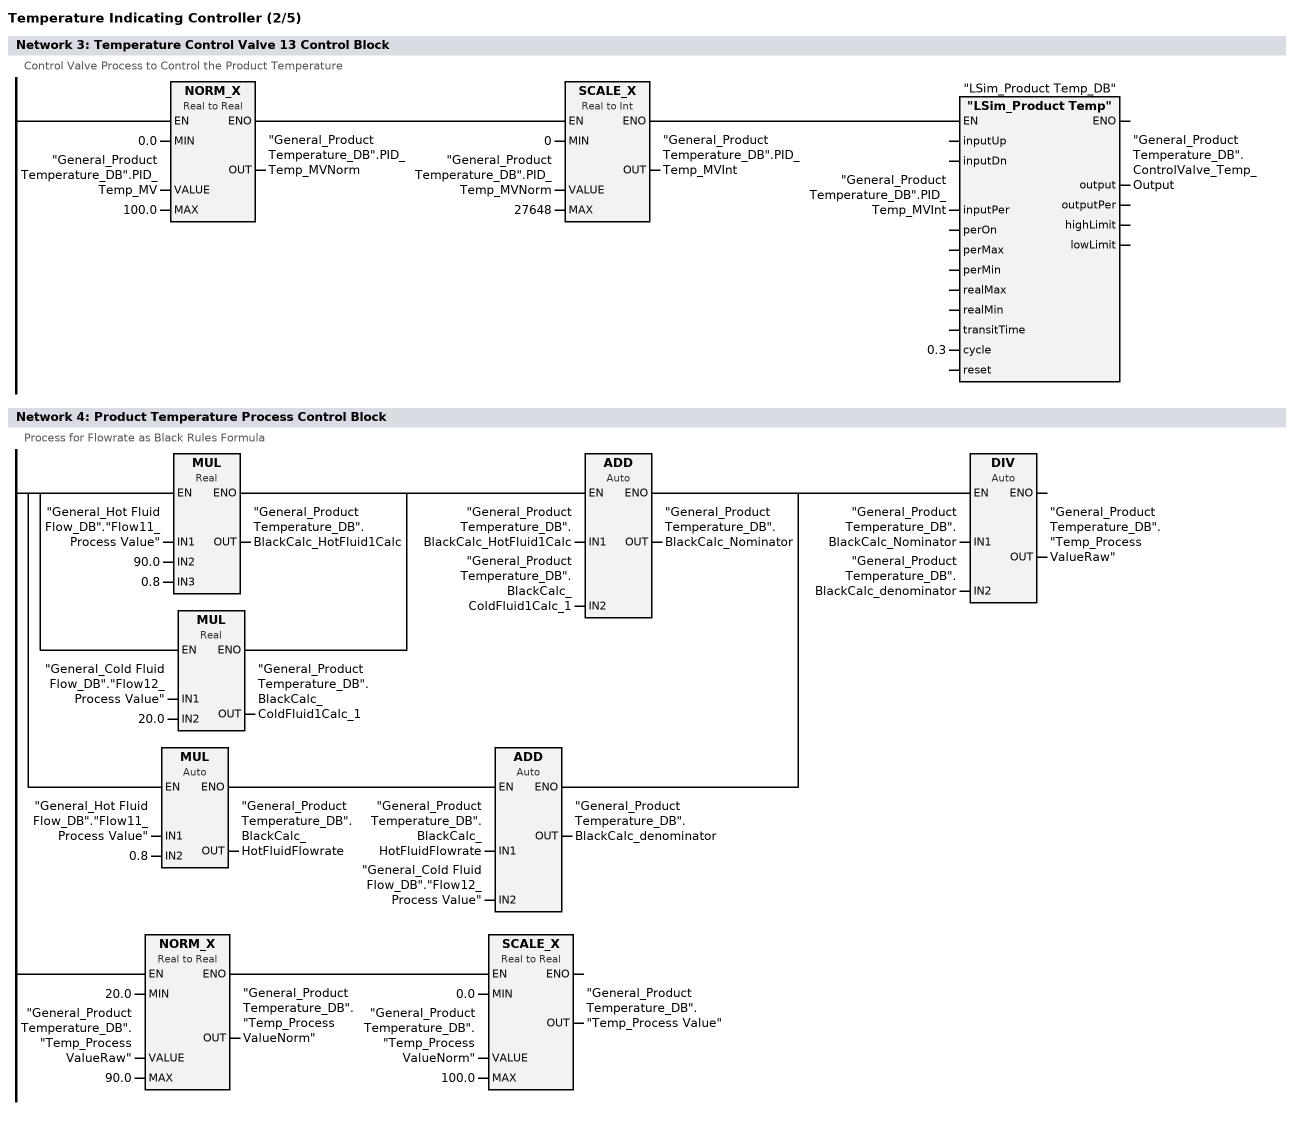
   RUNG wire#powerrail
      { S7_Templates := "[SrcType := Real, DestType := Real]" } Normalize(min := 0.0, value := "General_Product Temperature_DB".PID_Temp_MV, max := 100.0, out => "General_Product Temperature_DB".PID_Temp_MVNorm)
      { S7_Templates := "[SrcType := Real, DestType := Int]" } Scale(min := 0, value := "General_Product Temperature_DB".PID_Temp_MVNorm, max := 27648, out => "General_Product Temperature_DB".PID_Temp_MVInt)
      "LSim_Product Temp_DB"(inputUp :=, inputDn :=, inputPer := "General_Product Temperature_DB".PID_Temp_MVInt, perOn :=, perMax :=, perMin :=, realMax :=, realMin :=, transitTime :=, cycle := 0.3, reset :=, output => "General_Product Temperature_DB".ControlValve_Temp_Output, outputPer =>, highLimit =>, lowLimit =>)
   END_RUNG
   // the same network as SCL:
   "General_Product Temperature_DB".PID_Temp_MVNorm := NORM_X(MIN := 0.0, VALUE := "General_Product Temperature_DB".PID_Temp_MV, MAX := 100.0);
   "General_Product Temperature_DB".PID_Temp_MVInt := SCALE_X(MIN := 0, VALUE := "General_Product Temperature_DB".PID_Temp_MVNorm, MAX := 27648);
   "LSim_Product Temp_DB"(inputPer := "General_Product Temperature_DB".PID_Temp_MVInt,   // "LSim_Product Temp"
                          cycle := 0.3,
                          output => "General_Product Temperature_DB".ControlValve_Temp_Output);
END_REGION

REGION Network 4: Product Temperature Process Control Block
   // Process for Flowrate as Black Rules Formula
   RUNG wire#powerrail
      { S7_Templates := "SrcType := Real" } Mul(in1 := "General_Hot Fluid Flow_DB"."Flow11_Process Value", in2 := 90.0, in3 := 0.8, out => "General_Product Temperature_DB".BlackCalc_HotFluid1Calc)
      wire#w1
      Add(in1 := "General_Product Temperature_DB".BlackCalc_HotFluid1Calc, in2 := "General_Product Temperature_DB".BlackCalc_ColdFluid1Calc_1, out => "General_Product Temperature_DB".BlackCalc_Nominator)
      wire#w2
      Div(in1 := "General_Product Temperature_DB".BlackCalc_Nominator, in2 := "General_Product Temperature_DB".BlackCalc_denominator, out => "General_Product Temperature_DB"."Temp_Process ValueRaw")
   END_RUNG
   RUNG wire#powerrail
      { S7_Templates := "SrcType := Real" } Mul(in1 := "General_Cold Fluid Flow_DB"."Flow12_Process Value", in2 := 20.0, out => "General_Product Temperature_DB".BlackCalc_ColdFluid1Calc_1)
   END_RUNG wire#w1
   RUNG wire#powerrail
      Mul(in1 := "General_Hot Fluid Flow_DB"."Flow11_Process Value", in2 := 0.8, out => "General_Product Temperature_DB".BlackCalc_HotFluidFlowrate)
      Add(in1 := "General_Product Temperature_DB".BlackCalc_HotFluidFlowrate, in2 := "General_Cold Fluid Flow_DB"."Flow12_Process Value", out => "General_Product Temperature_DB".BlackCalc_denominator)
   END_RUNG wire#w2
   RUNG wire#powerrail
      { S7_Templates := "[SrcType := Real, DestType := Real]" } Normalize(min := 20.0, value := "General_Product Temperature_DB"."Temp_Process ValueRaw", max := 90.0, out => "General_Product Temperature_DB"."Temp_Process ValueNorm")
      { S7_Templates := "[SrcType := Real, DestType := Real]" } Scale(min := 0.0, value := "General_Product Temperature_DB"."Temp_Process ValueNorm", max := 100.0, out => "General_Product Temperature_DB"."Temp_Process Value")
   END_RUNG
   // the same network as SCL:
   "General_Product Temperature_DB".BlackCalc_HotFluid1Calc := "General_Hot Fluid Flow_DB"."Flow11_Process Value" * 90.0 * 0.8;
   "General_Product Temperature_DB".BlackCalc_ColdFluid1Calc_1 := "General_Cold Fluid Flow_DB"."Flow12_Process Value" * 20.0;
   IF TRUE OR TRUE THEN
       "General_Product Temperature_DB".BlackCalc_Nominator := "General_Product Temperature_DB".BlackCalc_HotFluid1Calc + "General_Product Temperature_DB".BlackCalc_ColdFluid1Calc_1;
   END_IF;
   "General_Product Temperature_DB".BlackCalc_HotFluidFlowrate := "General_Hot Fluid Flow_DB"."Flow11_Process Value" * 0.8;
   "General_Product Temperature_DB".BlackCalc_denominator := "General_Product Temperature_DB".BlackCalc_HotFluidFlowrate + "General_Cold Fluid Flow_DB"."Flow12_Process Value";
   IF TRUE OR TRUE OR TRUE THEN
       "General_Product Temperature_DB"."Temp_Process ValueRaw" := "General_Product Temperature_DB".BlackCalc_Nominator / "General_Product Temperature_DB".BlackCalc_denominator;
   END_IF;
   "General_Product Temperature_DB"."Temp_Process ValueNorm" := NORM_X(MIN := 20.0, VALUE := "General_Product Temperature_DB"."Temp_Process ValueRaw", MAX := 90.0);
   "General_Product Temperature_DB"."Temp_Process Value" := SCALE_X(MIN := 0.0, VALUE := "General_Product Temperature_DB"."Temp_Process ValueNorm", MAX := 100.0);
END_REGION

REGION Network 5: Safety Block For Temperature Limit
   // Set Alarm Limit for TSH and TSL activate when Level at 85 C and 20 C
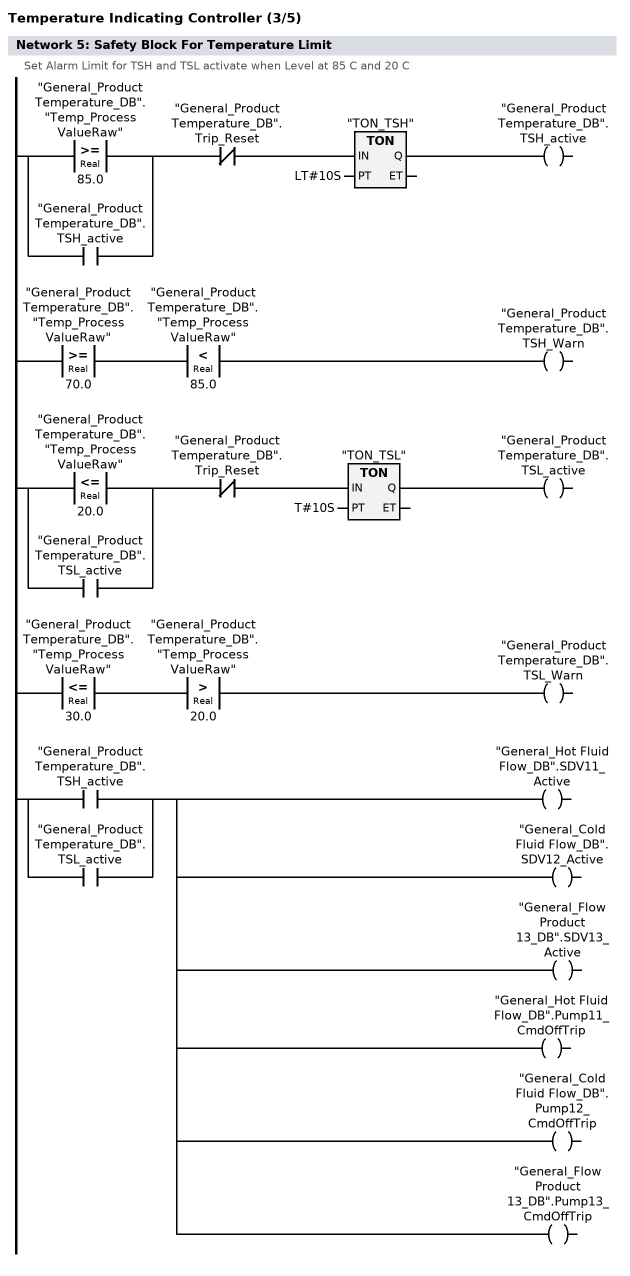
   "TON_TSH".TON(IN := (("General_Product Temperature_DB"."Temp_Process ValueRaw" >= 85.0) OR "General_Product Temperature_DB".TSH_active) AND NOT "General_Product Temperature_DB".Trip_Reset,
                 PT := LT#10S);
   "General_Product Temperature_DB".TSH_active := "TON_TSH".Q;
   "General_Product Temperature_DB".TSH_Warn := ("General_Product Temperature_DB"."Temp_Process ValueRaw" >= 70.0) AND ("General_Product Temperature_DB"."Temp_Process ValueRaw" < 85.0);
   "TON_TSL".TON(IN := (("General_Product Temperature_DB"."Temp_Process ValueRaw" <= 20.0) OR "General_Product Temperature_DB".TSL_active) AND NOT "General_Product Temperature_DB".Trip_Reset,
                 PT := T#10S);
   "General_Product Temperature_DB".TSL_active := "TON_TSL".Q;
   "General_Product Temperature_DB".TSL_Warn := ("General_Product Temperature_DB"."Temp_Process ValueRaw" <= 30.0) AND ("General_Product Temperature_DB"."Temp_Process ValueRaw" > 20.0);
   "General_Hot Fluid Flow_DB".SDV11_Active := "General_Product Temperature_DB".TSH_active OR "General_Product Temperature_DB".TSL_active;
   "General_Cold Fluid Flow_DB".SDV12_Active := "General_Hot Fluid Flow_DB".SDV11_Active;
   "General_Flow Product 13_DB".SDV13_Active := "General_Hot Fluid Flow_DB".SDV11_Active;
   "General_Hot Fluid Flow_DB".Pump11_CmdOffTrip := "General_Hot Fluid Flow_DB".SDV11_Active;
   "General_Cold Fluid Flow_DB".Pump12_CmdOffTrip := "General_Hot Fluid Flow_DB".SDV11_Active;
   "General_Flow Product 13_DB".Pump13_CmdOffTrip := "General_Hot Fluid Flow_DB".SDV11_Active;
END_REGION

REGION Network 6: Alarm Management Block
   // Control Block for Managing the Alarm Occured in the System
